C05439=1080.298,356.414,-96.423,176.101,28.139,154.837
C05440=1080.292,356.167,-96.387,176.097,28.133,154.836
C05441=1080.286,355.919,-96.351,176.094,28.128,154.835
C05442=1080.280,355.672,-96.316,176.091,28.123,154.834
C05443=1080.275,355.425,-96.280,176.087,28.117,154.833
C05444=1080.268,355.178,-96.244,176.084,28.111,154.832
C05445=1080.262,354.930,-96.209,176.081,28.106,154.831
C05446=1080.256,354.683,-96.173,176.078,28.100,154.830
C05447=1080.249,354.435,-96.137,176.074,28.095,154.829
C05448=1080.244,354.188,-96.102,176.071,28.089,154.828
C05449=1080.237,353.941,-96.067,176.068,28.083,154.827
C05450=1080.231,353.693,-96.031,176.065,28.078,154.826
C05451=1080.225,353.445,-95.995,176.061,28.073,154.825
C05452=1080.220,353.198,-95.960,176.058,28.067,154.824
C05453=1080.213,352.951,-95.925,176.055,28.062,154.823
C05454=1080.207,352.703,-95.889,176.052,28.056,154.822
C05455=1080.201,352.456,-95.853,176.048,28.051,154.821
C05456=1080.195,352.209,-95.818,176.045,28.045,154.820
C05457=1080.189,351.961,-95.783,176.041,28.040,154.820
C05458=1080.183,351.714,-95.747,176.038,28.035,154.819
C05459=1080.176,351.466,-95.712,176.034,28.029,154.818
C05460=1080.171,351.219,-95.676,176.031,28.024,154.817
C05461=1080.164,350.972,-95.641,176.028,28.019,154.816
C05462=1080.158,350.724,-95.606,176.025,28.013,154.815
C05463=1080.153,350.477,-95.571,176.022,28.008,154.814
C05464=1080.146,350.229,-95.536,176.018,28.002,154.813
C05465=1080.140,349.982,-95.500,176.015,27.997,154.812
C05466=1080.134,349.735,-95.465,176.012,27.992,154.811
C05467=1080.128,349.487,-95.430,176.009,27.987,154.810
C05468=1080.121,349.239,-95.395,176.005,27.981,154.809
C05469=1080.116,348.992,-95.360,176.002,27.976,154.808
C05470=1080.109,348.745,-95.325,175.999,27.971,154.807
C05471=1080.103,348.497,-95.290,175.995,27.965,154.807
C05472=1080.097,348.250,-95.255,175.992,27.960,154.806
C05473=1080.091,348.002,-95.219,175.989,27.955,154.805
C05474=1080.085,347.755,-95.185,175.985,27.950,154.804
C05475=1080.079,347.507,-95.149,175.982,27.944,154.803
C05476=1080.073,347.259,-95.115,175.979,27.939,154.802
C05477=1080.067,347.012,-95.080,175.976,27.934,154.801
C05478=1080.061,346.765,-95.044,175.973,27.929,154.800
C05479=1080.055,346.518,-95.010,175.970,27.924,154.799
C05480=1080.049,346.270,-94.975,175.966,27.918,154.798
C05481=1080.043,346.022,-94.940,175.963,27.913,154.797
C05482=1080.037,345.775,-94.905,175.959,27.908,154.797
C05483=1080.030,345.527,-94.870,175.956,27.903,154.796
C05484=1080.025,345.280,-94.835,175.953,27.898,154.795
C05485=1080.018,345.032,-94.801,175.950,27.893,154.794
C05486=1080.009,344.621,-94.743,175.945,27.884,154.793
C05487=1079.998,344.208,-94.686,175.939,27.876,154.791
C05488=1079.988,343.795,-94.628,175.934,27.867,154.790
C05489=1079.978,343.384,-94.570,175.928,27.858,154.788
C05490=1079.972,343.135,-94.535,175.925,27.854,154.787
C05491=1079.967,342.888,-94.501,175.922,27.848,154.786
C05492=1079.960,342.641,-94.466,175.919,27.843,154.786
C05493=1079.954,342.394,-94.432,175.916,27.839,154.785
C05494=1079.947,342.146,-94.397,175.912,27.833,154.784
C05495=1079.942,341.898,-94.363,175.909,27.828,154.783
C05496=1079.936,341.650,-94.328,175.906,27.823,154.782
C05497=1079.930,341.403,-94.294,175.903,27.818,154.781
C05498=1079.923,341.155,-94.259,175.899,27.813,154.781
C05499=1079.917,340.908,-94.225,175.896,27.808,154.780
C05500=1079.912,340.661,-94.191,175.893,27.803,154.779
C05501=1079.906,340.412,-94.156,175.890,27.798,154.778
C05502=1079.900,340.165,-94.122,175.887,27.793,154.777
C05503=1079.894,339.917,-94.087,175.884,27.788,154.776
C05504=1079.888,339.670,-94.053,175.881,27.784,154.775
C05505=1079.882,339.423,-94.019,175.877,27.778,154.775
C05506=1079.875,339.175,-93.985,175.874,27.773,154.774
C05507=1079.869,338.927,-93.951,175.871,27.768,154.773
C05508=1079.864,338.679,-93.916,175.867,27.763,154.772
C05509=1079.858,338.432,-93.882,175.864,27.758,154.771
C05510=1079.852,338.184,-93.848,175.861,27.754,154.770
C05511=1079.846,337.936,-93.813,175.858,27.748,154.770
C05512=1079.840,337.689,-93.779,175.855,27.744,154.769
C05513=1079.834,337.441,-93.746,175.852,27.739,154.768
C05514=1079.828,337.193,-93.712,175.849,27.734,154.767
C05515=1079.822,336.946,-93.678,175.846,27.729,154.766
C05516=1079.816,336.699,-93.643,175.843,27.724,154.766
C05517=1079.809,336.451,-93.609,175.839,27.720,154.765
C05518=1079.804,336.203,-93.575,175.836,27.715,154.764
C05519=1079.797,335.956,-93.542,175.833,27.710,154.763
C05520=1079.791,335.708,-93.508,175.830,27.705,154.762
C05521=1079.785,335.461,-93.474,175.827,27.700,154.762
C05522=1079.779,335.213,-93.440,175.824,27.695,154.761
C05523=1079.773,334.965,-93.406,175.821,27.691,154.760
C05524=1079.767,334.717,-93.372,175.818,27.685,154.759
C05525=1079.761,334.470,-93.338,175.815,27.681,154.758
C05526=1079.756,334.222,-93.305,175.811,27.676,154.758
C05527=1079.749,333.974,-93.270,175.807,27.671,154.757
C05528=1079.744,333.726,-93.237,175.804,27.666,154.756
C05529=1079.737,333.479,-93.203,175.801,27.662,154.755
C05530=1079.731,333.232,-93.169,175.798,27.656,154.754
C05531=1079.726,332.984,-93.136,175.795,27.652,154.754
C05532=1079.719,332.736,-93.102,175.792,27.647,154.753
C05533=1079.714,332.488,-93.068,175.789,27.642,154.752
C05534=1079.708,332.241,-93.034,175.786,27.638,154.751
C05535=1079.702,331.993,-93.001,175.783,27.633,154.750
C05536=1079.696,331.746,-92.967,175.780,27.628,154.750
C05537=1079.690,331.498,-92.934,175.777,27.624,154.749
C05538=1079.679,331.080,-92.877,175.772,27.615,154.748
C05539=1079.669,330.662,-92.821,175.766,27.608,154.746
C05540=1079.659,330.245,-92.765,175.760,27.600,154.745
C05541=1079.648,329.827,-92.708,175.756,27.592,154.744
C05542=1079.642,329.579,-92.674,175.753,27.588,154.743
C05543=1079.636,329.331,-92.642,175.750,27.583,154.742
C05544=1079.630,329.084,-92.608,175.746,27.579,154.742
C05545=1079.624,328.836,-92.575,175.743,27.574,154.741
C05546=1079.618,328.588,-92.542,175.740,27.569,154.740
C05547=1079.612,328.341,-92.509,175.737,27.565,154.739
C05548=1079.606,328.092,-92.475,175.734,27.560,154.739
C05549=1079.599,327.845,-92.442,175.731,27.555,154.738
C05550=1079.594,327.597,-92.408,175.728,27.551,154.737
C05551=1079.587,327.350,-92.376,175.725,27.546,154.736
C05552=1079.582,327.102,-92.342,175.721,27.542,154.736
C05553=1079.575,326.854,-92.310,175.718,27.537,154.735
C05554=1079.570,326.606,-92.276,175.715,27.533,154.734
C05555=1079.564,326.359,-92.243,175.712,27.528,154.733
C05556=1079.558,326.112,-92.209,175.709,27.523,154.733
C05557=1079.551,325.863,-92.176,175.707,27.519,154.732
C05558=1079.545,325.615,-92.143,175.704,27.515,154.731
C05559=1079.539,325.368,-92.110,175.700,27.510,154.730
C05560=1079.533,325.120,-92.077,175.697,27.506,154.730
C05561=1079.527,324.872,-92.044,175.694,27.501,154.729
C05562=1079.521,324.625,-92.011,175.691,27.497,154.728
C05563=1079.515,324.377,-91.978,175.688,27.492,154.728
C05564=1079.509,324.129,-91.945,175.685,27.487,154.727
C05565=1079.503,323.881,-91.912,175.682,27.483,154.726
C05566=1079.497,323.633,-91.880,175.678,27.478,154.725
C05567=1079.491,323.385,-91.847,175.676,27.474,154.725
C05568=1079.486,323.138,-91.814,175.673,27.469,154.724
C05569=1079.479,322.890,-91.781,175.670,27.465,154.723
C05570=1079.474,322.642,-91.748,175.667,27.460,154.723
C05571=1079.467,322.394,-91.715,175.664,27.456,154.722
C05572=1079.461,322.147,-91.682,175.660,27.451,154.721
C05573=1079.457,321.899,-91.650,175.657,27.447,154.720
C05574=1079.450,321.651,-91.617,175.654,27.442,154.720
C05575=1079.445,321.404,-91.584,175.651,27.438,154.719
C05576=1079.438,321.156,-91.551,175.649,27.434,154.718
C05577=1079.432,320.908,-91.518,175.646,27.429,154.717
C05578=1079.427,320.660,-91.486,175.643,27.425,154.717
C05579=1079.421,320.412,-91.453,175.639,27.420,154.716
C05580=1079.414,320.165,-91.420,175.636,27.416,154.715
C05581=1079.409,319.916,-91.388,175.633,27.411,154.715
C05582=1079.403,319.669,-91.355,175.630,27.407,154.714
C05583=1079.397,319.422,-91.323,175.628,27.402,154.713
C05584=1079.392,319.173,-91.290,175.625,27.398,154.713
C05585=1079.386,318.925,-91.257,175.622,27.393,154.712
C05586=1079.379,318.678,-91.225,175.618,27.389,154.711
C05587=1079.374,318.430,-91.193,175.615,27.384,154.710
C05588=1079.368,318.182,-91.160,175.612,27.380,154.710
C05589=1079.362,317.934,-91.128,175.610,27.376,154.709
C05590=1079.357,317.723,-91.099,175.607,27.372,154.708
C05591=1079.353,317.510,-91.072,175.605,27.368,154.708
C05592=1079.347,317.297,-91.044,175.602,27.364,154.707
C05593=1079.342,317.086,-91.015,175.599,27.360,154.707
C05594=1079.337,316.874,-90.988,175.597,27.356,154.706
C05595=1079.332,316.662,-90.961,175.594,27.353,154.705
C05596=1079.328,316.449,-90.933,175.592,27.349,154.705
C05597=1079.323,316.238,-90.905,175.589,27.345,154.704
C05598=1079.317,315.989,-90.873,175.587,27.341,154.703
C05599=1079.311,315.741,-90.841,175.584,27.337,154.703
C05600=1079.306,315.494,-90.808,175.580,27.332,154.702
C05601=1079.300,315.246,-90.776,175.577,27.327,154.701
C05602=1079.294,314.998,-90.743,175.574,27.323,154.701
C05603=1079.288,314.751,-90.711,175.572,27.319,154.700
C05604=1079.282,314.502,-90.679,175.569,27.314,154.699
C05605=1079.276,314.255,-90.646,175.566,27.310,154.699
C05606=1079.270,314.007,-90.614,175.562,27.306,154.698
C05607=1079.264,313.758,-90.582,175.559,27.302,154.697
C05608=1079.258,313.511,-90.551,175.556,27.297,154.697
C05609=1079.251,313.264,-90.519,175.554,27.293,154.696
C05610=1079.245,313.015,-90.487,175.551,27.289,154.695
C05611=1079.239,312.767,-90.455,175.548,27.285,154.695
C05612=1079.233,312.519,-90.422,175.544,27.281,154.694
C05613=1079.228,312.272,-90.391,175.541,27.276,154.694
C05614=1079.221,312.024,-90.359,175.539,27.272,154.693
C05615=1079.215,311.776,-90.327,175.536,27.268,154.692
C05616=1079.210,311.529,-90.295,175.533,27.264,154.692
C05617=1079.204,311.280,-90.263,175.530,27.260,154.691
C05618=1079.198,311.032,-90.231,175.527,27.256,154.690
C05619=1079.191,310.784,-90.200,175.524,27.251,154.690
C05620=1079.186,310.537,-90.168,175.521,27.247,154.689
C05621=1079.180,310.288,-90.136,175.518,27.243,154.688
C05622=1079.174,310.040,-90.104,175.515,27.238,154.688
C05623=1079.168,309.793,-90.073,175.512,27.234,154.687
C05624=1079.162,309.545,-90.041,175.509,27.230,154.686
C05625=1079.156,309.297,-90.009,175.506,27.226,154.686
C05626=1079.150,309.049,-89.977,175.503,27.222,154.685
C05627=1079.143,308.801,-89.946,175.501,27.218,154.684
C05628=1079.138,308.554,-89.914,175.498,27.213,154.684
C05629=1079.132,308.305,-89.882,175.494,27.209,154.683
C05630=1079.127,308.058,-89.850,175.491,27.205,154.682
C05631=1079.120,307.810,-89.819,175.488,27.201,154.682
C05632=1079.114,307.562,-89.787,175.486,27.197,154.681
C05633=1079.109,307.314,-89.755,175.483,27.193,154.681
C05634=1079.102,307.066,-89.724,175.480,27.188,154.680
C05635=1079.096,306.819,-89.692,175.476,27.184,154.679
C05636=1079.091,306.570,-89.661,175.474,27.180,154.679
C05637=1079.085,306.323,-89.630,175.471,27.176,154.678
C05638=1079.079,306.075,-89.598,175.468,27.172,154.677
C05639=1079.073,305.827,-89.566,175.465,27.167,154.677
C05640=1079.067,305.579,-89.535,175.463,27.163,154.676
C05641=1079.061,305.331,-89.504,175.459,27.159,154.675
C05642=1079.056,305.083,-89.472,175.456,27.155,154.675
C05643=1079.049,304.836,-89.440,175.454,27.151,154.674
C05644=1079.043,304.587,-89.408,175.451,27.147,154.674
C05645=1079.038,304.339,-89.378,175.448,27.143,154.673
C05646=1079.032,304.129,-89.351,175.445,27.139,154.672
C05647=1079.028,303.919,-89.324,175.443,27.136,154.672
C05648=1079.023,303.708,-89.297,175.441,27.132,154.671
C05649=1079.018,303.497,-89.271,175.437,27.128,154.671
C05650=1079.013,303.287,-89.244,175.435,27.125,154.670
C05651=1079.008,303.076,-89.217,175.433,27.121,154.670
C05652=1079.003,302.866,-89.192,175.431,27.118,154.669
C05653=1078.998,302.655,-89.164,175.428,27.115,154.669
C05654=1078.993,302.407,-89.133,175.425,27.110,154.668
C05655=1078.986,302.159,-89.102,175.422,27.106,154.667
C05656=1078.981,301.911,-89.071,175.420,27.102,154.667
C05657=1078.975,301.663,-89.040,175.417,27.098,154.666
C05658=1078.970,301.415,-89.009,175.413,27.094,154.666
C05659=1078.964,301.167,-88.977,175.411,27.090,154.665
C05660=1078.958,300.919,-88.946,175.408,27.086,154.664
C05661=1078.952,300.671,-88.915,175.405,27.081,154.664
C05662=1078.947,300.423,-88.884,175.403,27.077,154.663
C05663=1078.941,300.175,-88.852,175.400,27.073,154.662
C05664=1078.935,299.927,-88.822,175.396,27.069,154.662
C05665=1078.929,299.680,-88.790,175.394,27.065,154.661
C05666=1078.923,299.431,-88.759,175.391,27.061,154.661
C05667=1078.918,299.184,-88.728,175.388,27.057,154.660
C05668=1078.912,298.936,-88.697,175.385,27.052,154.659
C05669=1078.907,298.688,-88.666,175.383,27.048,154.659
C05670=1078.901,298.440,-88.634,175.379,27.044,154.658
C05671=1078.895,298.192,-88.604,175.377,27.040,154.657
C05672=1078.890,297.944,-88.573,175.374,27.036,154.657
C05673=1078.884,297.697,-88.542,175.371,27.032,154.656
C05674=1078.877,297.448,-88.511,175.369,27.028,154.656
C05675=1078.872,297.200,-88.480,175.365,27.024,154.655
C05676=1078.866,296.952,-88.450,175.362,27.020,154.654
C05677=1078.860,296.704,-88.419,175.360,27.016,154.654
C05678=1078.855,296.456,-88.388,175.357,27.012,154.653
C05679=1078.849,296.208,-88.357,175.354,27.008,154.652
C05680=1078.842,295.960,-88.327,175.351,27.004,154.652
C05681=1078.836,295.712,-88.296,175.348,27.000,154.651
C05682=1078.831,295.464,-88.265,175.345,26.996,154.651
C05683=1078.825,295.215,-88.235,175.343,26.992,154.650
C05684=1078.819,294.968,-88.204,175.340,26.988,154.649
C05685=1078.813,294.720,-88.173,175.337,26.984,154.649
C05686=1078.807,294.472,-88.143,175.334,26.980,154.648
C05687=1078.802,294.224,-88.112,175.331,26.976,154.648
C05688=1078.796,293.976,-88.081,175.328,26.972,154.647
C05689=1078.790,293.728,-88.051,175.326,26.968,154.647
C05690=1078.784,293.480,-88.020,175.323,26.964,154.646
C05691=1078.778,293.232,-87.990,175.320,26.960,154.645
C05692=1078.772,292.984,-87.959,175.317,26.956,154.645
C05693=1078.766,292.736,-87.929,175.314,26.952,154.644
C05694=1078.761,292.488,-87.898,175.312,26.948,154.644
C05695=1078.755,292.240,-87.868,175.309,26.944,154.643
C05696=1078.749,291.991,-87.837,175.306,26.940,154.642
C05697=1078.743,291.744,-87.807,175.303,26.936,154.642
C05698=1078.737,291.496,-87.776,175.300,26.932,154.641
C05699=1078.732,291.247,-87.747,175.298,26.928,154.641
C05700=1078.726,291.000,-87.716,175.295,26.924,154.640
C05701=1078.719,290.751,-87.686,175.292,26.920,154.639
C05702=1078.710,290.344,-87.636,175.288,26.914,154.639
C05703=1078.700,289.938,-87.586,175.283,26.907,154.638
C05704=1078.691,289.531,-87.536,175.279,26.901,154.637
C05705=1078.682,289.124,-87.487,175.274,26.894,154.636
C05706=1078.675,288.876,-87.456,175.271,26.891,154.635
C05707=1078.670,288.628,-87.427,175.268,26.887,154.635
C05708=1078.664,288.380,-87.396,175.265,26.883,154.634
C05709=1078.658,288.132,-87.366,175.262,26.879,154.633
C05710=1078.652,287.884,-87.337,175.260,26.875,154.633
C05711=1078.646,287.636,-87.307,175.257,26.871,154.632
C05712=1078.640,287.388,-87.276,175.254,26.868,154.632
C05713=1078.634,287.139,-87.246,175.251,26.863,154.631
C05714=1078.628,286.891,-87.216,175.249,26.860,154.631
C05715=1078.623,286.643,-87.186,175.246,26.856,154.630
C05716=1078.617,286.395,-87.156,175.243,26.852,154.629
C05717=1078.611,286.147,-87.126,175.240,26.848,154.629
C05718=1078.605,285.899,-87.097,175.237,26.844,154.628
C05719=1078.599,285.651,-87.066,175.235,26.840,154.628
C05720=1078.594,285.403,-87.037,175.232,26.836,154.627
C05721=1078.588,285.155,-87.006,175.230,26.832,154.627
C05722=1078.582,284.906,-86.977,175.226,26.828,154.626
C05723=1078.577,284.659,-86.946,175.224,26.825,154.625
C05724=1078.570,284.410,-86.917,175.221,26.821,154.625
C05725=1078.564,284.163,-86.887,175.218,26.817,154.624
C05726=1078.559,283.914,-86.857,175.216,26.813,154.624
C05727=1078.553,283.666,-86.827,175.213,26.809,154.623
C05728=1078.548,283.418,-86.797,175.210,26.805,154.623
C05729=1078.541,283.170,-86.767,175.207,26.801,154.622
C05730=1078.536,282.922,-86.738,175.205,26.798,154.621
C05731=1078.530,282.674,-86.708,175.202,26.794,154.621
C05732=1078.524,282.426,-86.678,175.200,26.790,154.620
C05733=1078.519,282.177,-86.648,175.196,26.786,154.620
C05734=1078.513,281.929,-86.619,175.194,26.782,154.619
C05735=1078.507,281.681,-86.589,175.191,26.778,154.619
C05736=1078.501,281.433,-86.559,175.189,26.774,154.618
C05737=1078.496,281.184,-86.529,175.186,26.770,154.617
C05738=1078.489,280.937,-86.500,175.182,26.766,154.617
C05739=1078.484,280.688,-86.470,175.180,26.763,154.616
C05740=1078.478,280.440,-86.440,175.177,26.758,154.616
C05741=1078.472,280.192,-86.411,175.175,26.755,154.615
C05742=1078.466,279.943,-86.382,175.172,26.751,154.615
C05743=1078.460,279.696,-86.352,175.169,26.747,154.614
C05744=1078.454,279.447,-86.322,175.166,26.743,154.614
C05745=1078.449,279.199,-86.293,175.164,26.740,154.613
C05746=1078.442,278.951,-86.264,175.161,26.736,154.613
C05747=1078.437,278.702,-86.234,175.159,26.732,154.612
C05748=1078.431,278.454,-86.205,175.155,26.728,154.611
C05749=1078.425,278.206,-86.175,175.153,26.724,154.611
C05750=1078.420,277.959,-86.145,175.150,26.720,154.610
C05751=1078.414,277.711,-86.116,175.148,26.717,154.610
C05752=1078.408,277.462,-86.087,175.145,26.713,154.609
C05753=1078.402,277.214,-86.058,175.142,26.709,154.609
C05754=1078.393,276.817,-86.011,175.138,26.703,154.608
C05755=1078.384,276.419,-85.964,175.134,26.697,154.607
C05756=1078.374,276.023,-85.917,175.129,26.691,154.606
C05757=1078.365,275.626,-85.870,175.125,26.685,154.605
C05758=1078.359,275.378,-85.841,175.122,26.681,154.605
C05759=1078.353,275.130,-85.812,175.120,26.677,154.604
C05760=1078.347,274.881,-85.782,175.117,26.673,154.603
C05761=1078.341,274.633,-85.753,175.115,26.670,154.603
C05762=1078.337,274.385,-85.725,175.112,26.666,154.602
C05763=1078.330,274.137,-85.696,175.109,26.662,154.602
C05764=1078.325,273.888,-85.666,175.106,26.658,154.601
C05765=1078.319,273.640,-85.637,175.104,26.654,154.601
C05766=1078.312,273.392,-85.608,175.101,26.651,154.600
C05767=1078.307,273.144,-85.579,175.099,26.647,154.600
C05768=1078.301,272.896,-85.550,175.095,26.643,154.599
C05769=1078.296,272.647,-85.521,175.093,26.639,154.599
C05770=1078.290,272.399,-85.492,175.090,26.635,154.598
C05771=1078.283,272.151,-85.463,175.088,26.632,154.597
C05772=1078.278,271.903,-85.435,175.085,26.628,154.597
C05773=1078.273,271.654,-85.405,175.082,26.624,154.596
C05774=1078.266,271.406,-85.376,175.080,26.621,154.596
C05775=1078.260,271.157,-85.348,175.077,26.617,154.595
C05776=1078.255,270.909,-85.318,175.075,26.613,154.595
C05777=1078.249,270.662,-85.289,175.072,26.609,154.594
C05778=1078.243,270.413,-85.261,175.069,26.605,154.594
C05779=1078.238,270.164,-85.231,175.066,26.602,154.593
C05780=1078.232,269.916,-85.202,175.064,26.598,154.593
C05781=1078.226,269.668,-85.174,175.061,26.594,154.592
C05782=1078.220,269.420,-85.145,175.059,26.591,154.592
C05783=1078.214,269.172,-85.116,175.056,26.587,154.591
C05784=1078.209,268.924,-85.088,175.053,26.583,154.590
C05785=1078.203,268.675,-85.059,175.051,26.579,154.590
C05786=1078.197,268.427,-85.030,175.048,26.575,154.589
C05787=1078.191,268.179,-85.001,175.046,26.572,154.589
C05788=1078.185,267.930,-84.973,175.042,26.568,154.588
C05789=1078.179,267.682,-84.944,175.040,26.564,154.588
C05790=1078.174,267.433,-84.916,175.037,26.561,154.587
C05791=1078.168,267.186,-84.887,175.035,26.557,154.587
C05792=1078.162,266.937,-84.859,175.033,26.553,154.586
C05793=1078.156,266.689,-84.829,175.029,26.550,154.586
C05794=1078.151,266.441,-84.802,175.027,26.545,154.585
C05795=1078.145,266.192,-84.773,175.024,26.542,154.585
C05796=1078.138,265.944,-84.744,175.022,26.538,154.584
C05797=1078.133,265.696,-84.716,175.020,26.535,154.584
C05798=1078.128,265.447,-84.687,175.016,26.531,154.583
C05799=1078.122,265.199,-84.658,175.014,26.527,154.583
C05800=1078.116,264.951,-84.630,175.011,26.523,154.582
C05801=1078.110,264.703,-84.601,175.009,26.520,154.581
C05802=1078.104,264.454,-84.573,175.007,26.516,154.581
C05803=1078.099,264.206,-84.545,175.004,26.512,154.580
C05804=1078.093,263.957,-84.517,175.001,26.508,154.580
C05805=1078.087,263.710,-84.488,174.998,26.504,154.579
C05806=1078.077,263.315,-84.443,174.994,26.499,154.579
C05807=1078.068,262.921,-84.399,174.991,26.493,154.578
C05808=1078.059,262.527,-84.354,174.986,26.487,154.577
C05809=1078.049,262.134,-84.309,174.982,26.481,154.576
C05810=1078.043,261.885,-84.281,174.979,26.478,154.576
C05811=1078.038,261.637,-84.253,174.977,26.474,154.575
C05812=1078.031,261.389,-84.225,174.974,26.470,154.575
C05813=1078.025,261.140,-84.197,174.971,26.467,154.574
C05814=1078.020,260.892,-84.168,174.969,26.463,154.573
C05815=1078.014,260.644,-84.140,174.966,26.459,154.573
C05816=1078.008,260.396,-84.112,174.964,26.456,154.573
C05817=1078.002,260.147,-84.084,174.961,26.453,154.572
C05818=1077.996,259.898,-84.056,174.958,26.449,154.572
C05819=1077.990,259.650,-84.028,174.956,26.445,154.571
C05820=1077.984,259.402,-83.999,174.954,26.442,154.570
C05821=1077.978,259.154,-83.972,174.951,26.438,154.570
C05822=1077.972,258.905,-83.944,174.948,26.434,154.569
C05823=1077.967,258.657,-83.916,174.945,26.430,154.569
C05824=1077.961,258.408,-83.887,174.943,26.427,154.568
C05825=1077.955,258.161,-83.860,174.941,26.423,154.568
C05826=1077.949,257.912,-83.832,174.938,26.419,154.567
C05827=1077.944,257.664,-83.804,174.935,26.416,154.567
C05828=1077.938,257.415,-83.775,174.933,26.412,154.566
C05829=1077.932,257.167,-83.749,174.930,26.408,154.566
C05830=1077.926,256.918,-83.720,174.928,26.405,154.565
C05831=1077.921,256.670,-83.692,174.926,26.401,154.565
C05832=1077.915,256.421,-83.664,174.922,26.397,154.564
C05833=1077.909,256.173,-83.637,174.920,26.394,154.564
C05834=1077.903,255.925,-83.608,174.918,26.390,154.563
C05835=1077.898,255.677,-83.580,174.915,26.386,154.563
C05836=1077.891,255.428,-83.553,174.913,26.383,154.562
C05837=1077.886,255.179,-83.525,174.910,26.379,154.562
C05838=1077.880,254.931,-83.497,174.907,26.375,154.561
C05839=1077.874,254.683,-83.470,174.905,26.372,154.561
C05840=1077.868,254.434,-83.442,174.903,26.368,154.560
C05841=1077.863,254.186,-83.414,174.900,26.364,154.560
C05842=1077.857,253.938,-83.387,174.897,26.360,154.559
C05843=1077.851,253.689,-83.358,174.895,26.357,154.559
C05844=1077.846,253.440,-83.331,174.892,26.353,154.558
C05845=1077.839,253.192,-83.304,174.890,26.349,154.557
C05846=1077.834,252.944,-83.276,174.888,26.346,154.557
C05847=1077.829,252.695,-83.248,174.885,26.342,154.556
C05848=1077.822,252.447,-83.221,174.882,26.338,154.556
C05849=1077.817,252.199,-83.193,174.880,26.335,154.555
C05850=1077.812,251.950,-83.165,174.877,26.331,154.555
C05851=1077.805,251.702,-83.138,174.875,26.327,154.554
C05852=1077.800,251.453,-83.110,174.873,26.324,154.554
C05853=1077.795,251.205,-83.082,174.869,26.320,154.553
C05854=1077.788,250.956,-83.055,174.867,26.316,154.553
C05855=1077.783,250.708,-83.027,174.865,26.313,154.552
C05856=1077.777,250.460,-83.000,174.862,26.309,154.552
C05857=1077.771,250.211,-82.973,174.860,26.305,154.551
C05858=1077.763,249.815,-82.928,174.856,26.299,154.550
C05859=1077.753,249.418,-82.885,174.852,26.293,154.549
C05860=1077.744,249.021,-82.841,174.848,26.287,154.549
C05861=1077.735,248.625,-82.798,174.844,26.281,154.548
C05862=1077.729,248.376,-82.770,174.842,26.278,154.547
C05863=1077.724,248.128,-82.743,174.840,26.274,154.547
C05864=1077.718,247.880,-82.715,174.836,26.270,154.546
C05865=1077.713,247.631,-82.688,174.834,26.267,154.546
C05866=1077.707,247.382,-82.661,174.832,26.263,154.545
C05867=1077.701,247.134,-82.633,174.829,26.259,154.545
C05868=1077.696,246.886,-82.606,174.827,26.255,154.544
C05869=1077.690,246.637,-82.579,174.825,26.252,154.544
C05870=1077.684,246.389,-82.551,174.822,26.248,154.543
C05871=1077.678,246.140,-82.525,174.819,26.244,154.543
C05872=1077.673,245.892,-82.497,174.817,26.241,154.542
C05873=1077.667,245.644,-82.470,174.815,26.237,154.542
C05874=1077.661,245.395,-82.443,174.813,26.234,154.541
C05875=1077.656,245.146,-82.416,174.809,26.230,154.541
C05876=1077.650,244.898,-82.389,174.807,26.226,154.540
C05877=1077.644,244.650,-82.362,174.805,26.223,154.539
C05878=1077.639,244.401,-82.334,174.802,26.219,154.539
C05879=1077.632,244.152,-82.307,174.800,26.215,154.538
C05880=1077.627,243.904,-82.281,174.798,26.211,154.538
C05881=1077.622,243.655,-82.253,174.795,26.208,154.537
C05882=1077.616,243.407,-82.227,174.792,26.204,154.537
C05883=1077.610,243.159,-82.199,174.790,26.200,154.536
C05884=1077.604,242.910,-82.172,174.788,26.197,154.536
C05885=1077.598,242.661,-82.145,174.786,26.193,154.535
C05886=1077.593,242.413,-82.119,174.783,26.189,154.535
C05887=1077.587,242.165,-82.092,174.780,26.186,154.534
C05888=1077.581,241.916,-82.065,174.778,26.183,154.534
C05889=1077.575,241.667,-82.038,174.776,26.179,154.533
C05890=1077.570,241.419,-82.011,174.773,26.175,154.533
C05891=1077.564,241.170,-81.984,174.771,26.171,154.532
C05892=1077.558,240.922,-81.958,174.768,26.168,154.532
C05893=1077.552,240.674,-81.931,174.766,26.164,154.531
C05894=1077.547,240.425,-81.904,174.763,26.160,154.531
C05895=1077.540,240.176,-81.877,174.761,26.157,154.530
C05896=1077.534,239.928,-81.851,174.759,26.153,154.530
C05897=1077.529,239.679,-81.824,174.756,26.150,154.529
C05898=1077.524,239.431,-81.797,174.754,26.146,154.529
C05899=1077.518,239.182,-81.770,174.751,26.142,154.528
C05900=1077.512,238.934,-81.744,174.749,26.139,154.528
C05901=1077.506,238.685,-81.717,174.747,26.135,154.527
C05902=1077.500,238.437,-81.690,174.744,26.132,154.527
C05903=1077.494,238.188,-81.663,174.741,26.128,154.526
C05904=1077.489,237.939,-81.637,174.739,26.124,154.526
C05905=1077.483,237.691,-81.611,174.737,26.121,154.525
C05906=1077.477,237.443,-81.584,174.735,26.117,154.525
C05907=1077.471,237.194,-81.557,174.733,26.113,154.524
C05908=1077.466,236.946,-81.531,174.729,26.110,154.524
C05909=1077.460,236.698,-81.504,174.727,26.106,154.523
C05910=1077.450,236.293,-81.461,174.724,26.100,154.522
C05911=1077.441,235.891,-81.418,174.720,26.094,154.521
C05912=1077.432,235.487,-81.376,174.715,26.088,154.521
C05913=1077.423,235.085,-81.333,174.712,26.082,154.520
C05914=1077.417,234.836,-81.306,174.709,26.079,154.519
C05915=1077.412,234.587,-81.280,174.707,26.075,154.519
C05916=1077.406,234.339,-81.253,174.705,26.071,154.518
C05917=1077.400,234.091,-81.227,174.703,26.068,154.518
C05918=1077.395,233.842,-81.201,174.700,26.064,154.517
C05919=1077.389,233.593,-81.174,174.698,26.060,154.517
C05920=1077.383,233.345,-81.147,174.695,26.057,154.516
C05921=1077.377,233.095,-81.121,174.693,26.053,154.516
C05922=1077.371,232.847,-81.094,174.691,26.050,154.515
C05923=1077.366,232.598,-81.069,174.688,26.046,154.515
C05924=1077.360,232.350,-81.043,174.686,26.042,154.514
C05925=1077.354,232.102,-81.016,174.684,26.039,154.514
C05926=1077.349,231.853,-80.990,174.681,26.035,154.513
C05927=1077.343,231.605,-80.964,174.679,26.032,154.513
C05928=1077.337,231.356,-80.938,174.676,26.028,154.512
C05929=1077.332,231.107,-80.911,174.674,26.024,154.512
C05930=1077.326,230.858,-80.885,174.672,26.020,154.511
C05931=1077.320,230.610,-80.859,174.670,26.017,154.511
C05932=1077.314,230.361,-80.833,174.667,26.013,154.510
C05933=1077.308,230.113,-80.807,174.665,26.010,154.510
C05934=1077.303,229.864,-80.781,174.662,26.006,154.509
C05935=1077.296,229.616,-80.755,174.660,26.002,154.509
C05936=1077.291,229.367,-80.729,174.658,25.998,154.508
C05937=1077.285,229.118,-80.703,174.656,25.995,154.508
C05938=1077.279,228.870,-80.677,174.653,25.992,154.507
C05939=1077.273,228.621,-80.651,174.651,25.988,154.507
C05940=1077.268,228.372,-80.625,174.648,25.984,154.506
C05941=1077.261,228.124,-80.599,174.646,25.981,154.506
C05942=1077.256,227.875,-80.573,174.644,25.977,154.505
C05943=1077.251,227.626,-80.547,174.642,25.973,154.504
C05944=1077.245,227.379,-80.521,174.639,25.970,154.504
C05945=1077.239,227.130,-80.495,174.637,25.966,154.503
C05946=1077.234,226.881,-80.469,174.635,25.963,154.503
C05947=1077.227,226.633,-80.443,174.632,25.959,154.503
C05948=1077.222,226.384,-80.417,174.630,25.955,154.502
C05949=1077.215,226.135,-80.392,174.628,25.952,154.502
C05950=1077.210,225.886,-80.366,174.625,25.948,154.501
C05951=1077.204,225.638,-80.339,174.623,25.945,154.500
C05952=1077.199,225.390,-80.314,174.621,25.941,154.500
C05953=1077.193,225.141,-80.288,174.619,25.937,154.499
C05954=1077.187,224.892,-80.263,174.616,25.933,154.499
C05955=1077.182,224.643,-80.237,174.614,25.930,154.498
C05956=1077.176,224.395,-80.211,174.611,25.926,154.498
C05957=1077.170,224.146,-80.185,174.609,25.922,154.497
C05958=1077.165,223.898,-80.160,174.607,25.919,154.497
C05959=1077.158,223.649,-80.134,174.605,25.915,154.496
C05960=1077.153,223.400,-80.108,174.603,25.912,154.496
C05961=1077.148,223.151,-80.082,174.601,25.908,154.495
C05962=1077.138,222.740,-80.040,174.596,25.902,154.494
C05963=1077.129,222.328,-79.998,174.592,25.896,154.494
C05964=1077.119,221.917,-79.956,174.589,25.890,154.493
C05965=1077.110,221.506,-79.913,174.585,25.884,154.492
C05966=1077.104,221.257,-79.888,174.583,25.881,154.491
C05967=1077.098,221.008,-79.862,174.581,25.877,154.491
C05968=1077.092,220.759,-79.836,174.579,25.873,154.490
C05969=1077.086,220.510,-79.811,174.577,25.870,154.490
C05970=1077.081,220.262,-79.786,174.573,25.866,154.489
C05971=1077.075,220.013,-79.760,174.571,25.862,154.489
C05972=1077.069,219.765,-79.735,174.569,25.858,154.488
C05973=1077.063,219.516,-79.709,174.567,25.855,154.488
C05974=1077.058,219.268,-79.684,174.565,25.851,154.487
C05975=1077.052,219.019,-79.658,174.563,25.848,154.487
C05976=1077.045,218.770,-79.633,174.560,25.844,154.486
C05977=1077.040,218.521,-79.608,174.558,25.841,154.486
C05978=1077.035,218.273,-79.583,174.556,25.837,154.485
C05979=1077.028,218.024,-79.558,174.554,25.833,154.485
C05980=1077.023,217.775,-79.532,174.551,25.830,154.484
C05981=1077.017,217.527,-79.507,174.549,25.826,154.484
C05982=1077.011,217.279,-79.481,174.547,25.822,154.483
C05983=1077.006,217.029,-79.456,174.544,25.819,154.483
C05984=1077.000,216.780,-79.431,174.542,25.815,154.482
C05985=1076.994,216.532,-79.406,174.540,25.811,154.482
C05986=1076.988,216.284,-79.380,174.538,25.808,154.481
C05987=1076.983,216.034,-79.355,174.536,25.804,154.481
C05988=1076.977,215.786,-79.330,174.534,25.800,154.480
C05989=1076.971,215.537,-79.305,174.532,25.797,154.480
C05990=1076.966,215.289,-79.279,174.529,25.793,154.479
C05991=1076.960,215.040,-79.255,174.527,25.790,154.479
C05992=1076.954,214.791,-79.229,174.525,25.786,154.478
C05993=1076.948,214.543,-79.204,174.522,25.782,154.478
C05994=1076.943,214.294,-79.179,174.520,25.778,154.477
C05995=1076.937,214.045,-79.154,174.518,25.775,154.477
C05996=1076.931,213.797,-79.129,174.516,25.771,154.476
C05997=1076.926,213.548,-79.104,174.513,25.767,154.475
C05998=1076.921,213.299,-79.079,174.511,25.764,154.475
C05999=1076.914,213.051,-79.053,174.509,25.760,154.474
C06000=1076.909,212.801,-79.029,174.507,25.757,154.474
C06001=1076.903,212.553,-79.004,174.505,25.753,154.474
C06002=1076.897,212.304,-78.979,174.503,25.750,154.473
C06003=1076.891,212.056,-78.954,174.501,25.746,154.472
C06004=1076.886,211.807,-78.930,174.498,25.742,154.472
C06005=1076.879,211.558,-78.904,174.496,25.739,154.471
C06006=1076.875,211.309,-78.879,174.494,25.735,154.471
C06007=1076.869,211.061,-78.854,174.492,25.731,154.470
C06008=1076.863,210.812,-78.830,174.490,25.728,154.470
C06009=1076.857,210.563,-78.804,174.488,25.724,154.469
C06010=1076.852,210.315,-78.780,174.486,25.720,154.469
C06011=1076.846,210.066,-78.755,174.483,25.717,154.468
C06012=1076.840,209.817,-78.730,174.480,25.713,154.468
C06013=1076.834,209.569,-78.705,174.478,25.709,154.467
C06014=1076.825,209.161,-78.665,174.475,25.703,154.466
C06015=1076.816,208.754,-78.624,174.472,25.698,154.466
C06016=1076.806,208.347,-78.584,174.468,25.692,154.465
C06017=1076.796,207.939,-78.543,174.465,25.686,154.464
C06018=1076.773,206.902,-78.443,174.351,25.626,154.464
C06019=1076.768,206.653,-78.419,174.349,25.623,154.464
C06020=1076.761,206.404,-78.395,174.347,25.620,154.464
C06021=1076.756,206.156,-78.370,174.344,25.618,154.464
C06022=1076.750,205.907,-78.346,174.343,25.615,154.463
C06023=1076.745,205.658,-78.323,174.341,25.613,154.463
C06024=1076.739,205.409,-78.299,174.338,25.610,154.463
C06025=1076.734,205.160,-78.274,174.336,25.607,154.462
C06026=1076.728,204.912,-78.250,174.334,25.604,154.462
C06027=1076.722,204.664,-78.226,174.331,25.602,154.462
C06028=1076.717,204.414,-78.202,174.329,25.599,154.462
C06029=1076.711,204.165,-78.178,174.326,25.596,154.461
C06030=1076.705,203.917,-78.155,174.324,25.594,154.461
C06031=1076.700,203.668,-78.130,174.322,25.591,154.461
C06032=1076.695,203.419,-78.107,174.319,25.588,154.460
C06033=1076.688,203.170,-78.083,174.317,25.586,154.460
C06034=1076.683,202.921,-78.058,174.315,25.583,154.460
C06035=1076.678,202.673,-78.034,174.312,25.580,154.459
C06036=1076.672,202.424,-78.011,174.310,25.577,154.459
C06037=1076.667,202.175,-77.987,174.308,25.575,154.459
C06038=1076.660,201.926,-77.963,174.306,25.572,154.459
C06039=1076.654,201.677,-77.940,174.304,25.570,154.458
C06040=1076.649,201.429,-77.916,174.301,25.567,154.458
C06041=1076.643,201.180,-77.893,174.299,25.565,154.458
C06042=1076.637,200.931,-77.868,174.297,25.562,154.457
C06043=1076.631,200.682,-77.845,174.294,25.559,154.457
C06044=1076.626,200.433,-77.821,174.292,25.556,154.457
C06045=1076.620,200.185,-77.797,174.290,25.554,154.457
C06046=1076.615,199.936,-77.774,174.287,25.551,154.456
C06047=1076.609,199.687,-77.750,174.285,25.549,154.456
C06048=1076.603,199.438,-77.727,174.283,25.546,154.456
C06049=1076.598,199.189,-77.703,174.281,25.544,154.455
C06050=1076.592,198.941,-77.679,174.279,25.541,154.455
C06051=1076.586,198.692,-77.656,174.276,25.538,154.455
C06052=1076.580,198.443,-77.631,174.274,25.536,154.455
C06053=1076.574,198.194,-77.608,174.271,25.533,154.454
C06054=1076.569,197.945,-77.585,174.269,25.531,154.454
C06055=1076.563,197.696,-77.561,174.267,25.528,154.454
C06056=1076.558,197.448,-77.538,174.264,25.525,154.454
C06057=1076.552,197.199,-77.514,174.263,25.523,154.453
C06058=1076.547,196.950,-77.491,174.261,25.520,154.453
C06059=1076.540,196.702,-77.467,174.258,25.517,154.453
C06060=1076.535,196.452,-77.443,174.256,25.515,154.452
C06061=1076.529,196.204,-77.420,174.253,25.512,154.452
C06062=1076.523,195.955,-77.397,174.251,25.510,154.452
C06063=1076.518,195.705,-77.373,174.249,25.507,154.452
C06064=1076.512,195.457,-77.350,174.246,25.504,154.451
C06065=1076.506,195.208,-77.327,174.245,25.502,154.451
C06066=1076.501,194.959,-77.303,174.243,25.499,154.451
C06067=1076.495,194.711,-77.280,174.240,25.496,154.450
C06068=1076.490,194.462,-77.257,174.238,25.494,154.450
C06069=1076.485,194.213,-77.233,174.236,25.491,154.450
C06070=1076.479,193.964,-77.209,174.233,25.488,154.450
C06071=1076.473,193.716,-77.186,174.232,25.486,154.449
C06072=1076.468,193.466,-77.163,174.229,25.484,154.449
C06073=1076.462,193.217,-77.140,174.227,25.481,154.449
C06074=1076.456,192.969,-77.116,174.225,25.478,154.449
C06075=1076.450,192.719,-77.092,174.222,25.476,154.448
C06076=1076.445,192.470,-77.069,174.220,25.473,154.448
C06077=1076.439,192.221,-77.046,174.218,25.470,154.448
C06078=1076.433,191.973,-77.023,174.216,25.468,154.447
C06079=1076.427,191.692,-76.997,174.213,25.465,154.447
C06080=1076.421,191.412,-76.970,174.211,25.462,154.447
C06081=1076.415,191.131,-76.945,174.208,25.459,154.446
C06082=1076.409,190.850,-76.918,174.206,25.456,154.446
C06083=1076.403,190.602,-76.895,174.204,25.453,154.446
C06084=1076.397,190.353,-76.872,174.201,25.451,154.445
C06085=1076.391,190.104,-76.848,174.199,25.448,154.445
C06086=1076.386,189.855,-76.825,174.197,25.446,154.445
C06087=1076.381,189.606,-76.802,174.195,25.443,154.445
C06088=1076.375,189.357,-76.779,174.193,25.440,154.444
C06089=1076.369,189.109,-76.756,174.190,25.437,154.444
C06090=1076.365,188.860,-76.733,174.188,25.435,154.444
C06091=1076.359,188.611,-76.710,174.187,25.432,154.443
C06092=1076.353,188.362,-76.687,174.184,25.430,154.443
C06093=1076.348,188.113,-76.664,174.182,25.427,154.443
C06094=1076.343,187.864,-76.640,174.180,25.424,154.443
C06095=1076.337,187.615,-76.617,174.177,25.421,154.442
C06096=1076.331,187.366,-76.595,174.176,25.419,154.442
C06097=1076.325,187.117,-76.572,174.173,25.416,154.442
C06098=1076.320,186.869,-76.549,174.171,25.414,154.441
C06099=1076.315,186.620,-76.525,174.169,25.411,154.441
C06100=1076.310,186.371,-76.503,174.167,25.408,154.441
C06101=1076.304,186.122,-76.480,174.165,25.406,154.441
C06102=1076.298,185.873,-76.457,174.163,25.403,154.440
C06103=1076.292,185.624,-76.434,174.160,25.401,154.440
C06104=1076.287,185.375,-76.410,174.158,25.398,154.440
C06105=1076.282,185.126,-76.387,174.156,25.396,154.439
C06106=1076.276,184.878,-76.365,174.154,25.393,154.439
C06107=1076.271,184.629,-76.342,174.152,25.390,154.439
C06108=1076.265,184.380,-76.319,174.149,25.388,154.439
C06109=1076.260,184.131,-76.297,174.148,25.386,154.438
C06110=1076.253,183.882,-76.274,174.146,25.383,154.438
C06111=1076.247,183.633,-76.251,174.143,25.380,154.438
C06112=1076.242,183.384,-76.228,174.141,25.378,154.438
C06113=1076.236,183.136,-76.205,174.139,25.375,154.437
C06114=1076.230,182.887,-76.182,174.137,25.373,154.437
C06115=1076.224,182.637,-76.161,174.135,25.370,154.437
C06116=1076.218,182.389,-76.138,174.132,25.367,154.436
C06117=1076.213,182.140,-76.115,174.131,25.365,154.436
C06118=1076.207,181.891,-76.092,174.128,25.363,154.436
C06119=1076.200,181.642,-76.070,174.126,25.360,154.436
C06120=1076.195,181.393,-76.047,174.124,25.358,154.436
C06121=1076.189,181.144,-76.024,174.122,25.356,154.435
C06122=1076.184,180.896,-76.002,174.120,25.353,154.435
C06123=1076.178,180.646,-75.980,174.117,25.350,154.435
C06124=1076.172,180.397,-75.957,174.115,25.348,154.434
C06125=1076.166,180.149,-75.934,174.114,25.345,154.434
C06126=1076.161,179.900,-75.911,174.111,25.343,154.434
C06127=1076.155,179.650,-75.890,174.109,25.340,154.434
C06128=1076.149,179.402,-75.867,174.107,25.338,154.433
C06129=1076.144,179.153,-75.844,174.105,25.335,154.433
C06130=1076.138,178.904,-75.822,174.103,25.333,154.433
C06131=1076.132,178.655,-75.800,174.100,25.330,154.433
C06132=1076.126,178.406,-75.777,174.098,25.327,154.432
C06133=1076.121,178.157,-75.754,174.097,25.325,154.432
C06134=1076.115,177.908,-75.731,174.094,25.322,154.432
C06135=1076.109,177.659,-75.710,174.092,25.320,154.431
C06136=1076.104,177.411,-75.687,174.090,25.318,154.431
C06137=1076.098,177.161,-75.665,174.088,25.315,154.431
C06138=1076.092,176.912,-75.643,174.086,25.312,154.431
C06139=1076.086,176.664,-75.620,174.083,25.310,154.430
C06140=1076.081,176.415,-75.598,174.082,25.307,154.430
C06141=1076.075,176.166,-75.575,174.080,25.305,154.430
C06142=1076.069,175.917,-75.553,174.077,25.302,154.430
C06143=1076.063,175.636,-75.528,174.075,25.299,154.429
C06144=1076.057,175.355,-75.503,174.073,25.296,154.429
C06145=1076.050,175.074,-75.478,174.070,25.294,154.429
C06146=1076.044,174.793,-75.452,174.068,25.291,154.428
C06147=1076.038,174.544,-75.430,174.066,25.288,154.428
C06148=1076.032,174.295,-75.408,174.064,25.286,154.428
C06149=1076.027,174.046,-75.386,174.062,25.283,154.428
C06150=1076.021,173.797,-75.363,174.059,25.281,154.427
C06151=1076.015,173.548,-75.341,174.058,25.279,154.427
C06152=1076.010,173.299,-75.319,174.056,25.275,154.427
C06153=1076.005,173.050,-75.296,174.053,25.273,154.426
C06154=1075.999,172.801,-75.275,174.052,25.270,154.426
C06155=1075.993,172.553,-75.252,174.050,25.268,154.426
C06156=1075.988,172.303,-75.230,174.047,25.265,154.426
C06157=1075.982,172.054,-75.208,174.046,25.263,154.425
C06158=1075.976,171.805,-75.185,174.043,25.260,154.425
C06159=1075.971,171.556,-75.164,174.041,25.258,154.425
C06160=1075.965,171.307,-75.142,174.040,25.255,154.424
C06161=1075.960,171.059,-75.119,174.037,25.253,154.424
C06162=1075.954,170.810,-75.098,174.035,25.250,154.424
C06163=1075.948,170.560,-75.076,174.034,25.248,154.424
C06164=1075.943,170.312,-75.053,174.031,25.245,154.423
C06165=1075.937,170.063,-75.031,174.029,25.243,154.423
C06166=1075.932,169.813,-75.009,174.027,25.240,154.423
C06167=1075.927,169.565,-74.987,174.025,25.238,154.423
C06168=1075.920,169.316,-74.965,174.023,25.235,154.422
C06169=1075.915,169.067,-74.943,174.021,25.233,154.422
C06170=1075.909,168.818,-74.921,174.019,25.229,154.422
C06171=1075.904,168.568,-74.899,174.017,25.227,154.421
C06172=1075.898,168.321,-74.877,174.015,25.225,154.421
C06173=1075.893,168.071,-74.855,174.013,25.222,154.421
C06174=1075.888,167.822,-74.833,174.011,25.220,154.420
C06175=1075.882,167.573,-74.811,174.009,25.217,154.420
C06176=1075.876,167.324,-74.789,174.007,25.214,154.420
C06177=1075.871,167.075,-74.768,174.005,25.212,154.420
C06178=1075.865,166.826,-74.745,174.003,25.209,154.419
C06179=1075.859,166.578,-74.724,174.001,25.207,154.419
C06180=1075.854,166.328,-74.701,173.999,25.204,154.419
C06181=1075.849,166.079,-74.680,173.997,25.201,154.418
C06182=1075.843,165.830,-74.658,173.996,25.199,154.418
C06183=1075.838,165.581,-74.636,173.993,25.196,154.418
C06184=1075.832,165.332,-74.614,173.991,25.194,154.418
C06185=1075.827,165.083,-74.593,173.989,25.191,154.417
C06186=1075.821,164.834,-74.571,173.987,25.189,154.417
C06187=1075.816,164.586,-74.548,173.985,25.186,154.417
C06188=1075.810,164.337,-74.527,173.983,25.183,154.416
C06189=1075.805,164.088,-74.505,173.981,25.181,154.416
C06190=1075.799,163.839,-74.483,173.980,25.178,154.416
C06191=1075.794,163.590,-74.461,173.977,25.176,154.416
C06192=1075.788,163.341,-74.440,173.975,25.173,154.415
C06193=1075.783,163.092,-74.418,173.973,25.171,154.415
C06194=1075.777,162.843,-74.396,173.971,25.168,154.415
C06195=1075.772,162.594,-74.374,173.970,25.165,154.414
C06196=1075.766,162.345,-74.353,173.968,25.163,154.414
C06197=1075.761,162.096,-74.331,173.965,25.160,154.414
C06198=1075.755,161.847,-74.309,173.964,25.158,154.414
C06199=1075.750,161.598,-74.287,173.961,25.155,154.413
C06200=1075.744,161.348,-74.266,173.960,25.153,154.413
C06201=1075.739,161.099,-74.245,173.958,25.150,154.413
C06202=1075.733,160.850,-74.223,173.955,25.147,154.412
C06203=1075.728,160.601,-74.202,173.954,25.145,154.412
C06204=1075.721,160.352,-74.180,173.951,25.143,154.412
C06205=1075.717,160.103,-74.158,173.950,25.140,154.412
C06206=1075.710,159.854,-74.137,173.948,25.138,154.411
C06207=1075.704,159.573,-74.112,173.946,25.134,154.411
C06208=1075.698,159.291,-74.088,173.943,25.132,154.411
C06209=1075.691,159.010,-74.064,173.941,25.129,154.410
C06210=1075.685,158.729,-74.040,173.939,25.126,154.410
C06211=1075.679,158.480,-74.018,173.937,25.124,154.410
C06212=1075.674,158.231,-73.998,173.935,25.121,154.410
C06213=1075.668,157.982,-73.976,173.933,25.119,154.409
C06214=1075.663,157.733,-73.954,173.931,25.116,154.409
C06215=1075.657,157.484,-73.933,173.930,25.114,154.409
C06216=1075.651,157.235,-73.911,173.927,25.111,154.408
C06217=1075.645,156.985,-73.891,173.925,25.108,154.408
C06218=1075.640,156.737,-73.869,173.924,25.106,154.408
C06219=1075.634,156.488,-73.848,173.921,25.103,154.408
C06220=1075.629,156.238,-73.826,173.920,25.101,154.407
C06221=1075.623,155.990,-73.805,173.918,25.098,154.407
C06222=1075.617,155.741,-73.784,173.916,25.096,154.407
C06223=1075.612,155.492,-73.762,173.914,25.093,154.406
C06224=1075.606,155.242,-73.741,173.912,25.091,154.406
C06225=1075.600,154.994,-73.720,173.910,25.088,154.406
C06226=1075.594,154.745,-73.698,173.908,25.085,154.406
C06227=1075.589,154.495,-73.678,173.906,25.083,154.405
C06228=1075.583,154.247,-73.657,173.904,25.080,154.405
C06229=1075.577,153.998,-73.635,173.903,25.078,154.405
C06230=1075.572,153.749,-73.614,173.900,25.075,154.404
C06231=1075.566,153.499,-73.593,173.899,25.073,154.404
C06232=1075.561,153.250,-73.572,173.896,25.071,154.404
C06233=1075.555,153.002,-73.551,173.895,25.068,154.404
C06234=1075.549,152.753,-73.529,173.893,25.066,154.403
C06235=1075.544,152.503,-73.509,173.891,25.063,154.403
C06236=1075.537,152.254,-73.487,173.889,25.061,154.403
C06237=1075.533,152.005,-73.466,173.887,25.058,154.403
C06238=1075.527,151.756,-73.445,173.885,25.056,154.402
C06239=1075.521,151.507,-73.424,173.883,25.053,154.402
C06240=1075.516,151.258,-73.403,173.881,25.051,154.402
C06241=1075.511,151.009,-73.382,173.879,25.048,154.401
C06242=1075.504,150.760,-73.361,173.878,25.046,154.401
C06243=1075.498,150.511,-73.340,173.875,25.043,154.401
C06244=1075.493,150.262,-73.319,173.874,25.040,154.401
C06245=1075.487,150.013,-73.298,173.872,25.038,154.400
C06246=1075.481,149.764,-73.277,173.870,25.035,154.400
C06247=1075.476,149.515,-73.256,173.868,25.033,154.400
C06248=1075.470,149.266,-73.235,173.866,25.030,154.399
C06249=1075.465,149.017,-73.214,173.864,25.028,154.399
C06250=1075.459,148.768,-73.193,173.863,25.025,154.399
C06251=1075.453,148.518,-73.172,173.860,25.023,154.399
C06252=1075.448,148.269,-73.151,173.859,25.020,154.398
C06253=1075.443,148.021,-73.130,173.857,25.018,154.398
C06254=1075.437,147.771,-73.109,173.855,25.015,154.398
C06255=1075.430,147.523,-73.089,173.853,25.013,154.398
C06256=1075.425,147.273,-73.068,173.851,25.010,154.397
C06257=1075.419,147.024,-73.047,173.849,25.008,154.397
C06258=1075.414,146.775,-73.026,173.848,25.005,154.397
C06259=1075.408,146.526,-73.005,173.845,25.003,154.396
C06260=1075.402,146.277,-72.985,173.844,25.000,154.396
C06261=1075.396,146.028,-72.964,173.842,24.998,154.396
C06262=1075.391,145.779,-72.943,173.840,24.995,154.396
C06263=1075.385,145.529,-72.922,173.838,24.993,154.395
C06264=1075.379,145.281,-72.902,173.836,24.991,154.395
C06265=1075.374,145.032,-72.881,173.834,24.987,154.395
C06266=1075.368,144.783,-72.860,173.833,24.985,154.394
C06267=1075.363,144.533,-72.840,173.831,24.982,154.394
C06268=1075.357,144.284,-72.818,173.829,24.980,154.394
C06269=1075.351,144.035,-72.798,173.827,24.977,154.394
C06270=1075.346,143.786,-72.778,173.825,24.975,154.393
C06271=1075.339,143.505,-72.754,173.823,24.972,154.393
C06272=1075.333,143.223,-72.731,173.821,24.969,154.393
C06273=1075.326,142.941,-72.708,173.819,24.967,154.392
C06274=1075.319,142.660,-72.684,173.817,24.964,154.392
C06275=1075.314,142.410,-72.664,173.815,24.961,154.392
C06276=1075.309,142.161,-72.643,173.814,24.959,154.391
C06277=1075.304,141.912,-72.623,173.811,24.956,154.391
C06278=1075.297,141.663,-72.602,173.810,24.954,154.391
C06279=1075.292,141.414,-72.581,173.807,24.951,154.391
C06280=1075.286,141.165,-72.560,173.806,24.949,154.390
C06281=1075.280,140.916,-72.540,173.804,24.946,154.390
C06282=1075.275,140.667,-72.520,173.802,24.943,154.390
C06283=1075.270,140.418,-72.499,173.800,24.941,154.389
C06284=1075.263,140.169,-72.479,173.799,24.938,154.389
C06285=1075.258,139.919,-72.458,173.796,24.936,154.389
C06286=1075.253,139.670,-72.438,173.795,24.933,154.389
C06287=1075.246,139.422,-72.417,173.793,24.931,154.388
C06288=1075.241,139.172,-72.396,173.791,24.928,154.388
C06289=1075.235,138.923,-72.376,173.790,24.926,154.388
C06290=1075.229,138.674,-72.356,173.787,24.923,154.387
C06291=1075.224,138.425,-72.335,173.786,24.921,154.387
C06292=1075.218,138.176,-72.315,173.784,24.918,154.387
C06293=1075.213,137.927,-72.295,173.782,24.916,154.387
C06294=1075.206,137.678,-72.274,173.780,24.913,154.386
C06295=1075.201,137.429,-72.254,173.779,24.910,154.386
C06296=1075.195,137.180,-72.234,173.776,24.908,154.386
C06297=1075.190,136.931,-72.213,173.775,24.905,154.385
C06298=1075.184,136.682,-72.193,173.774,24.903,154.385
C06299=1075.178,136.433,-72.173,173.771,24.900,154.385
C06300=1075.172,136.183,-72.153,173.770,24.898,154.385
C06301=1075.167,135.934,-72.132,173.768,24.895,154.384
C06302=1075.161,135.685,-72.113,173.766,24.893,154.384
C06303=1075.156,135.436,-72.092,173.764,24.890,154.384
C06304=1075.150,135.187,-72.072,173.762,24.888,154.383
C06305=1075.144,134.938,-72.052,173.760,24.885,154.383
C06306=1075.138,134.689,-72.032,173.759,24.883,154.383
C06307=1075.133,134.440,-72.011,173.757,24.880,154.382
C06308=1075.127,134.190,-71.991,173.755,24.878,154.382
C06309=1075.121,133.941,-71.970,173.754,24.875,154.382
C06310=1075.115,133.692,-71.950,173.751,24.873,154.382
C06311=1075.110,133.442,-71.930,173.750,24.870,154.381
C06312=1075.104,133.194,-71.910,173.748,24.868,154.381
C06313=1075.099,132.945,-71.890,173.746,24.865,154.381
C06314=1075.093,132.696,-71.870,173.745,24.862,154.380
C06315=1075.088,132.447,-71.849,173.743,24.860,154.380
C06316=1075.082,132.197,-71.830,173.741,24.857,154.380
C06317=1075.077,131.948,-71.810,173.739,24.855,154.380
C06318=1075.070,131.699,-71.789,173.737,24.852,154.379
C06319=1075.064,131.450,-71.769,173.736,24.850,154.379
C06320=1075.058,131.201,-71.749,173.734,24.847,154.379
C06321=1075.053,130.951,-71.730,173.732,24.845,154.378
C06322=1075.047,130.702,-71.710,173.730,24.842,154.378
C06323=1075.041,130.454,-71.690,173.729,24.840,154.378
C06324=1075.036,130.204,-71.670,173.726,24.837,154.378
C06325=1075.030,129.955,-71.650,173.725,24.835,154.377
C06326=1075.024,129.706,-71.630,173.723,24.833,154.377
C06327=1075.018,129.457,-71.610,173.721,24.830,154.377
C06328=1075.012,129.207,-71.590,173.720,24.828,154.377
C06329=1075.006,128.958,-71.570,173.717,24.825,154.376
C06330=1075.001,128.709,-71.550,173.716,24.823,154.376
C06331=1074.995,128.460,-71.531,173.715,24.820,154.376
C06332=1074.989,128.211,-71.511,173.712,24.817,154.375
C06333=1074.983,127.962,-71.491,173.711,24.815,154.375
C06334=1074.978,127.713,-71.471,173.709,24.812,154.375
C06335=1074.971,127.430,-71.449,173.707,24.810,154.374
C06336=1074.965,127.150,-71.426,173.705,24.807,154.374
C06337=1074.958,126.868,-71.404,173.703,24.804,154.374
C06338=1074.951,126.586,-71.382,173.702,24.801,154.373
C06339=1074.945,126.337,-71.362,173.699,24.799,154.373
C06340=1074.940,126.087,-71.342,173.698,24.796,154.373
C06341=1074.934,125.838,-71.322,173.696,24.794,154.373
C06342=1074.929,125.589,-71.303,173.694,24.791,154.372
C06343=1074.923,125.340,-71.283,173.693,24.789,154.372
C06344=1074.917,125.091,-71.263,173.690,24.786,154.372
C06345=1074.911,124.842,-71.243,173.689,24.783,154.371
C06346=1074.906,124.593,-71.223,173.688,24.781,154.371
C06347=1074.900,124.343,-71.204,173.685,24.778,154.371
C06348=1074.894,124.094,-71.184,173.684,24.776,154.371
C06349=1074.888,123.845,-71.164,173.682,24.773,154.370
C06350=1074.883,123.597,-71.145,173.680,24.771,154.370
C06351=1074.877,123.347,-71.126,173.679,24.769,154.370
C06352=1074.872,123.098,-71.106,173.677,24.765,154.369
C06353=1074.866,122.849,-71.086,173.675,24.763,154.369
C06354=1074.861,122.599,-71.067,173.674,24.761,154.369
C06355=1074.855,122.351,-71.047,173.672,24.758,154.369
C06356=1074.849,122.101,-71.027,173.670,24.756,154.368
C06357=1074.843,121.852,-71.007,173.668,24.753,154.368
C06358=1074.837,121.603,-70.988,173.667,24.750,154.368
C06359=1074.832,121.353,-70.968,173.665,24.748,154.367
C06360=1074.826,121.104,-70.948,173.663,24.745,154.367
C06361=1074.821,120.855,-70.929,173.662,24.743,154.367
C06362=1074.815,120.606,-70.909,173.660,24.741,154.366
C06363=1074.809,120.357,-70.890,173.658,24.738,154.366
C06364=1074.804,120.108,-70.871,173.657,24.735,154.366
C06365=1074.798,119.859,-70.851,173.655,24.733,154.365
C06366=1074.792,119.610,-70.832,173.653,24.730,154.365
C06367=1074.787,119.360,-70.813,173.652,24.728,154.365
C06368=1074.781,119.111,-70.793,173.650,24.725,154.365
C06369=1074.776,118.862,-70.773,173.648,24.722,154.364
C06370=1074.770,118.612,-70.753,173.647,24.720,154.364
C06371=1074.764,118.363,-70.734,173.644,24.717,154.364
C06372=1074.759,118.115,-70.715,173.643,24.715,154.363
C06373=1074.753,117.865,-70.695,173.642,24.712,154.363
C06374=1074.747,117.616,-70.676,173.639,24.709,154.363
C06375=1074.741,117.367,-70.656,173.638,24.707,154.362
C06376=1074.736,117.118,-70.637,173.637,24.704,154.362
C06377=1074.730,116.868,-70.618,173.634,24.701,154.362
C06378=1074.725,116.619,-70.599,173.633,24.699,154.362
C06379=1074.719,116.371,-70.579,173.632,24.697,154.361
C06380=1074.713,116.121,-70.560,173.629,24.694,154.361
C06381=1074.708,115.872,-70.540,173.628,24.691,154.361
C06382=1074.702,115.622,-70.521,173.627,24.689,154.360
C06383=1074.698,115.373,-70.502,173.624,24.686,154.360
C06384=1074.692,115.124,-70.482,173.623,24.683,154.360
C06385=1074.686,114.875,-70.462,173.622,24.681,154.359
C06386=1074.680,114.626,-70.443,173.619,24.678,154.359
C06387=1074.675,114.376,-70.424,173.618,24.676,154.359
C06388=1074.669,114.127,-70.405,173.617,24.673,154.358
C06389=1074.663,113.878,-70.386,173.614,24.670,154.358
C06390=1074.657,113.629,-70.367,173.613,24.668,154.358
C06391=1074.651,113.380,-70.347,173.612,24.666,154.358
C06392=1074.646,113.131,-70.328,173.609,24.663,154.357
C06393=1074.640,112.881,-70.309,173.608,24.660,154.357
C06394=1074.635,112.632,-70.290,173.607,24.658,154.357
C06395=1074.629,112.383,-70.271,173.604,24.655,154.356
C06396=1074.623,112.134,-70.252,173.603,24.653,154.356
C06397=1074.617,111.884,-70.233,173.602,24.650,154.356
C06398=1074.611,111.635,-70.214,173.599,24.647,154.355
C06399=1074.605,111.354,-70.192,173.598,24.645,154.355
C06400=1074.599,111.072,-70.171,173.596,24.641,154.355
C06401=1074.592,110.790,-70.149,173.595,24.639,154.354
C06402=1074.586,110.509,-70.127,173.592,24.636,154.354
C06403=1074.579,110.259,-70.108,173.591,24.634,154.354
C06404=1074.573,110.010,-70.089,173.589,24.631,154.353
C06405=1074.569,109.761,-70.071,173.587,24.628,154.353
C06406=1074.563,109.511,-70.052,173.586,24.626,154.353
C06407=1074.557,109.262,-70.033,173.584,24.623,154.353
C06408=1074.551,109.013,-70.014,173.582,24.621,154.352
C06409=1074.545,108.763,-69.995,173.581,24.618,154.352
C06410=1074.539,108.515,-69.976,173.580,24.616,154.352
C06411=1074.534,108.265,-69.957,173.577,24.613,154.351
C06412=1074.528,108.016,-69.938,173.576,24.610,154.351
C06413=1074.522,107.767,-69.919,173.575,24.608,154.351
C06414=1074.516,107.518,-69.900,173.572,24.605,154.350
C06415=1074.511,107.269,-69.881,173.571,24.603,154.350
C06416=1074.504,107.019,-69.862,173.570,24.600,154.350
C06417=1074.499,106.770,-69.843,173.567,24.597,154.349
C06418=1074.494,106.521,-69.825,173.566,24.595,154.349
C06419=1074.487,106.272,-69.806,173.565,24.593,154.349
C06420=1074.482,106.022,-69.787,173.563,24.589,154.349
C06421=1074.477,105.773,-69.768,173.561,24.587,154.348
C06422=1074.470,105.524,-69.750,173.560,24.585,154.348
C06423=1074.465,105.275,-69.730,173.558,24.582,154.348
C06424=1074.459,105.025,-69.712,173.556,24.579,154.347
C06425=1074.453,104.776,-69.694,173.555,24.577,154.347
C06426=1074.448,104.527,-69.674,173.553,24.574,154.347
C06427=1074.442,104.278,-69.655,173.551,24.572,154.346
C06428=1074.436,104.029,-69.637,173.550,24.569,154.346
C06429=1074.431,103.779,-69.618,173.549,24.567,154.346
C06430=1074.425,103.530,-69.599,173.547,24.564,154.345
C06431=1074.419,103.281,-69.581,173.545,24.561,154.345
C06432=1074.414,103.032,-69.561,173.544,24.559,154.345
C06433=1074.407,102.782,-69.544,173.542,24.556,154.344
C06434=1074.402,102.533,-69.525,173.540,24.554,154.344
C06435=1074.397,102.284,-69.505,173.539,24.551,154.344
C06436=1074.390,102.035,-69.487,173.537,24.548,154.344
C06437=1074.385,101.785,-69.469,173.536,24.546,154.343
C06438=1074.380,101.536,-69.449,173.534,24.543,154.343
C06439=1074.374,101.288,-69.431,173.532,24.540,154.343
C06440=1074.369,101.037,-69.413,173.531,24.538,154.342
C06441=1074.362,100.788,-69.394,173.529,24.535,154.342
C06442=1074.356,100.539,-69.375,173.527,24.533,154.342
C06443=1074.351,100.290,-69.357,173.526,24.530,154.341
C06444=1074.344,100.041,-69.338,173.525,24.528,154.341
C06445=1074.339,99.791,-69.319,173.522,24.525,154.341
C06446=1074.333,99.542,-69.302,173.521,24.523,154.341
C06447=1074.328,99.293,-69.282,173.520,24.520,154.340
C06448=1074.321,99.043,-69.264,173.518,24.517,154.340
C06449=1074.316,98.795,-69.246,173.516,24.515,154.340
C06450=1074.310,98.545,-69.227,173.515,24.512,154.339
C06451=1074.304,98.296,-69.209,173.513,24.510,154.339
C06452=1074.299,98.047,-69.190,173.511,24.507,154.339
C06453=1074.293,97.797,-69.172,173.510,24.504,154.338
C06454=1074.287,97.549,-69.154,173.508,24.502,154.338
C06455=1074.281,97.299,-69.135,173.507,24.500,154.338
C06456=1074.275,97.049,-69.117,173.505,24.497,154.337
C06457=1074.270,96.801,-69.098,173.504,24.494,154.337
C06458=1074.264,96.551,-69.080,173.502,24.492,154.337
C06459=1074.258,96.303,-69.062,173.501,24.489,154.336
C06460=1074.253,96.053,-69.043,173.499,24.486,154.336
C06461=1074.246,95.803,-69.024,173.497,24.484,154.336
C06462=1074.241,95.554,-69.007,173.496,24.482,154.336
C06463=1074.235,95.272,-68.986,173.494,24.478,154.335
C06464=1074.228,94.991,-68.965,173.493,24.475,154.335
C06465=1074.222,94.709,-68.944,173.490,24.473,154.335
C06466=1074.215,94.427,-68.924,173.489,24.470,154.334
C06467=1074.209,94.178,-68.905,173.487,24.467,154.334
C06468=1074.204,93.929,-68.887,173.486,24.464,154.333
C06469=1074.197,93.680,-68.869,173.484,24.462,154.333
C06470=1074.192,93.430,-68.850,173.483,24.459,154.333
C06471=1074.186,93.181,-68.833,173.481,24.456,154.332
C06472=1074.180,92.932,-68.814,173.479,24.454,154.332
C06473=1074.175,92.682,-68.796,173.478,24.452,154.332
C06474=1074.169,92.434,-68.777,173.477,24.449,154.331
C06475=1074.163,92.184,-68.760,173.474,24.446,154.331
C06476=1074.158,91.935,-68.741,173.473,24.444,154.331
C06477=1074.152,91.686,-68.723,173.472,24.441,154.331
C06478=1074.146,91.437,-68.705,173.470,24.438,154.330
C06479=1074.141,91.186,-68.687,173.468,24.436,154.330
C06480=1074.135,90.938,-68.668,173.467,24.433,154.330
C06481=1074.129,90.688,-68.650,173.466,24.430,154.329
C06482=1074.124,90.439,-68.633,173.464,24.428,154.329
C06483=1074.117,90.190,-68.614,173.462,24.425,154.329
C06484=1074.112,89.940,-68.596,173.461,24.422,154.328
C06485=1074.106,89.691,-68.578,173.459,24.420,154.328
C06486=1074.100,89.441,-68.560,173.458,24.418,154.328
C06487=1074.094,89.193,-68.542,173.457,24.415,154.327
C06488=1074.088,88.943,-68.524,173.454,24.412,154.327
C06489=1074.083,88.694,-68.506,173.453,24.410,154.327
C06490=1074.077,88.444,-68.488,173.452,24.407,154.327
C06491=1074.071,88.196,-68.470,173.450,24.405,154.326
C06492=1074.065,87.946,-68.452,173.448,24.402,154.326
C06493=1074.060,87.697,-68.434,173.447,24.399,154.326
C06494=1074.054,87.447,-68.416,173.445,24.397,154.325
C06495=1074.048,87.198,-68.399,173.444,24.395,154.325
C06496=1074.042,86.949,-68.380,173.442,24.391,154.325
C06497=1074.036,86.700,-68.362,173.441,24.389,154.324
C06498=1074.030,86.450,-68.344,173.439,24.387,154.324
C06499=1074.025,86.201,-68.327,173.438,24.384,154.324
C06500=1074.018,85.951,-68.309,173.436,24.381,154.323
C06501=1074.013,85.703,-68.291,173.434,24.379,154.323
C06502=1074.007,85.454,-68.273,173.433,24.376,154.323
C06503=1074.001,85.204,-68.255,173.432,24.373,154.322
C06504=1073.995,84.955,-68.238,173.430,24.371,154.322
C06505=1073.989,84.705,-68.220,173.428,24.368,154.322
C06506=1073.985,84.456,-68.201,173.427,24.366,154.321
C06507=1073.978,84.206,-68.184,173.425,24.363,154.321
C06508=1073.973,83.957,-68.166,173.424,24.361,154.321
C06509=1073.967,83.708,-68.148,173.422,24.358,154.321
C06510=1073.961,83.458,-68.130,173.421,24.355,154.320
C06511=1073.955,83.210,-68.112,173.419,24.353,154.320
C06512=1073.949,82.960,-68.094,173.418,24.350,154.320
C06513=1073.944,82.711,-68.077,173.417,24.348,154.319
C06514=1073.938,82.462,-68.059,173.414,24.345,154.319
C06515=1073.932,82.212,-68.041,173.413,24.342,154.319
C06516=1073.927,81.963,-68.024,173.412,24.340,154.318
C06517=1073.921,81.714,-68.006,173.410,24.337,154.318
C06518=1073.915,81.465,-67.988,173.409,24.334,154.318
C06519=1073.910,81.216,-67.971,173.407,24.332,154.317
C06520=1073.903,80.966,-67.953,173.406,24.329,154.317
C06521=1073.898,80.717,-67.935,173.404,24.326,154.317
C06522=1073.892,80.467,-67.917,173.403,24.324,154.316
C06523=1073.886,80.218,-67.900,173.401,24.321,154.316
C06524=1073.881,79.969,-67.882,173.399,24.318,154.316
C06525=1073.875,79.719,-67.864,173.398,24.316,154.315
C06526=1073.869,79.470,-67.846,173.397,24.313,154.315
C06527=1073.863,79.188,-67.827,173.395,24.310,154.315
C06528=1073.856,78.907,-67.807,173.393,24.307,154.314
C06529=1073.850,78.625,-67.787,173.391,24.304,154.314
C06530=1073.843,78.343,-67.767,173.390,24.301,154.314
C06531=1073.838,78.094,-67.750,173.389,24.299,154.313
C06532=1073.832,77.845,-67.732,173.387,24.296,154.313
C06533=1073.825,77.595,-67.715,173.385,24.293,154.313
C06534=1073.820,77.346,-67.697,173.384,24.291,154.312
C06535=1073.814,77.097,-67.680,173.382,24.289,154.312
C06536=1073.808,76.847,-67.662,173.381,24.286,154.312
C06537=1073.803,76.598,-67.644,173.379,24.283,154.311
C06538=1073.798,76.349,-67.627,173.378,24.281,154.311
C06539=1073.791,76.099,-67.610,173.376,24.278,154.311
C06540=1073.785,75.850,-67.593,173.375,24.275,154.310
C06541=1073.780,75.601,-67.575,173.374,24.273,154.310
C06542=1073.773,75.351,-67.557,173.372,24.270,154.310
C06543=1073.768,75.102,-67.541,173.370,24.267,154.309
C06544=1073.762,74.853,-67.523,173.369,24.265,154.309
C06545=1073.756,74.603,-67.505,173.368,24.262,154.309
C06546=1073.750,74.354,-67.488,173.366,24.260,154.308
C06547=1073.745,74.105,-67.470,173.364,24.257,154.308
C06548=1073.738,73.855,-67.454,173.363,24.254,154.308
C06549=1073.733,73.606,-67.436,173.361,24.252,154.307
C06550=1073.727,73.357,-67.418,173.360,24.249,154.307
C06551=1073.722,73.107,-67.402,173.359,24.246,154.307
C06552=1073.715,72.858,-67.384,173.357,24.244,154.307
C06553=1073.710,72.609,-67.367,173.355,24.241,154.306
C06554=1073.704,72.360,-67.349,173.354,24.238,154.306
C06555=1073.698,72.110,-67.332,173.353,24.236,154.306
C06556=1073.692,71.861,-67.315,173.351,24.234,154.305
C06557=1073.687,71.612,-67.297,173.350,24.231,154.305
C06558=1073.681,71.362,-67.280,173.348,24.228,154.305
C06559=1073.674,71.113,-67.263,173.347,24.225,154.304
C06560=1073.669,70.864,-67.246,173.345,24.223,154.304
C06561=1073.664,70.614,-67.229,173.344,24.220,154.304
C06562=1073.658,70.365,-67.211,173.343,24.217,154.303
C06563=1073.651,70.116,-67.194,173.340,24.215,154.303
C06564=1073.646,69.866,-67.177,173.339,24.212,154.303
C06565=1073.641,69.617,-67.159,173.338,24.209,154.302
C06566=1073.635,69.367,-67.143,173.337,24.207,154.302
C06567=1073.629,69.118,-67.125,173.335,24.205,154.302
C06568=1073.622,68.869,-67.108,173.333,24.201,154.301
C06569=1073.617,68.619,-67.091,173.332,24.199,154.301
C06570=1073.612,68.370,-67.074,173.330,24.197,154.301
C06571=1073.606,68.121,-67.058,173.329,24.194,154.300
C06572=1073.600,67.871,-67.040,173.328,24.191,154.300
C06573=1073.594,67.622,-67.023,173.326,24.189,154.300
C06574=1073.588,67.373,-67.006,173.324,24.186,154.299
C06575=1073.583,67.123,-66.989,173.323,24.183,154.299
C06576=1073.576,66.874,-66.972,173.322,24.181,154.299
C06577=1073.570,66.625,-66.954,173.320,24.178,154.298
C06578=1073.565,66.375,-66.938,173.319,24.176,154.298
C06579=1073.559,66.126,-66.920,173.318,24.173,154.298
C06580=1073.553,65.877,-66.904,173.316,24.170,154.297
C06581=1073.547,65.627,-66.887,173.314,24.168,154.297
C06582=1073.541,65.378,-66.870,173.313,24.165,154.297
C06583=1073.536,65.128,-66.853,173.312,24.162,154.296
C06584=1073.530,64.879,-66.836,173.310,24.160,154.296
C06585=1073.524,64.630,-66.819,173.308,24.157,154.296
C06586=1073.517,64.380,-66.802,173.307,24.154,154.296
C06587=1073.512,64.131,-66.785,173.306,24.152,154.295
C06588=1073.506,63.882,-66.768,173.304,24.150,154.295
C06589=1073.500,63.633,-66.752,173.303,24.147,154.295
C06590=1073.495,63.383,-66.735,173.302,24.144,154.294
C06591=1073.488,63.101,-66.716,173.300,24.141,154.294
C06592=1073.480,62.819,-66.697,173.298,24.139,154.294
C06593=1073.474,62.538,-66.677,173.296,24.135,154.293
C06594=1073.467,62.256,-66.658,173.295,24.132,154.293
C06595=1073.461,62.006,-66.642,173.294,24.130,154.293
C06596=1073.456,61.757,-66.625,173.291,24.127,154.292
C06597=1073.450,61.508,-66.608,173.290,24.125,154.292
C06598=1073.444,61.259,-66.592,173.289,24.122,154.292
C06599=1073.438,61.008,-66.575,173.287,24.120,154.291
C06600=1073.432,60.760,-66.558,173.286,24.117,154.291
C06601=1073.426,60.510,-66.541,173.285,24.114,154.291
C06602=1073.420,60.261,-66.525,173.283,24.112,154.290
C06603=1073.414,60.012,-66.508,173.281,24.109,154.290
C06604=1073.408,59.762,-66.491,173.280,24.107,154.290
C06605=1073.402,59.512,-66.475,173.279,24.104,154.289
C06606=1073.396,59.263,-66.457,173.277,24.102,154.289
C06607=1073.390,59.014,-66.441,173.276,24.099,154.289
C06608=1073.384,58.765,-66.425,173.274,24.096,154.288
C06609=1073.378,58.515,-66.408,173.273,24.094,154.288
C06610=1073.373,58.266,-66.391,173.271,24.091,154.288
C06611=1073.367,58.017,-66.375,173.270,24.088,154.287
C06612=1073.360,57.767,-66.358,173.269,24.086,154.287
C06613=1073.355,57.517,-66.341,173.267,24.083,154.287
C06614=1073.349,57.268,-66.325,173.266,24.081,154.287
C06615=1073.343,57.019,-66.308,173.264,24.078,154.286
C06616=1073.337,56.770,-66.292,173.262,24.075,154.286
C06617=1073.332,56.520,-66.275,173.261,24.073,154.286
C06618=1073.326,56.271,-66.258,173.260,24.070,154.285
C06619=1073.320,56.021,-66.242,173.259,24.068,154.285
C06620=1073.314,55.773,-66.225,173.257,24.065,154.285
C06621=1073.308,55.523,-66.208,173.255,24.062,154.284
C06622=1073.302,55.274,-66.192,173.254,24.060,154.284
C06623=1073.296,55.024,-66.176,173.252,24.057,154.284
C06624=1073.290,54.774,-66.159,173.251,24.054,154.283
C06625=1073.285,54.525,-66.142,173.250,24.052,154.283
C06626=1073.279,54.275,-66.126,173.249,24.050,154.283
C06627=1073.273,54.026,-66.110,173.246,24.046,154.282
C06628=1073.267,53.777,-66.094,173.245,24.044,154.282
C06629=1073.261,53.528,-66.077,173.244,24.041,154.282
C06630=1073.255,53.278,-66.060,173.243,24.039,154.281
C06631=1073.249,53.029,-66.044,173.241,24.036,154.281
C06632=1073.243,52.780,-66.027,173.240,24.033,154.281
C06633=1073.238,52.530,-66.011,173.239,24.031,154.280
C06634=1073.232,52.281,-65.995,173.236,24.028,154.280
C06635=1073.226,52.031,-65.978,173.235,24.025,154.280
C06636=1073.220,51.782,-65.962,173.234,24.023,154.279
C06637=1073.214,51.532,-65.945,173.233,24.021,154.279
C06638=1073.209,51.283,-65.929,173.231,24.018,154.279
C06639=1073.203,51.034,-65.913,173.230,24.015,154.278
C06640=1073.197,50.784,-65.896,173.229,24.012,154.278
C06641=1073.191,50.535,-65.880,173.227,24.010,154.278
C06642=1073.185,50.285,-65.864,173.225,24.007,154.278
C06643=1073.180,50.036,-65.847,173.224,24.004,154.277
C06644=1073.174,49.787,-65.831,173.223,24.002,154.277
C06645=1073.168,49.537,-65.814,173.222,23.999,154.276
C06646=1073.162,49.288,-65.798,173.220,23.997,154.276
C06647=1073.156,49.038,-65.782,173.219,23.994,154.276
C06648=1073.150,48.789,-65.765,173.217,23.991,154.275
C06649=1073.145,48.540,-65.750,173.215,23.989,154.275
C06650=1073.139,48.291,-65.733,173.214,23.986,154.275
C06651=1073.134,48.041,-65.717,173.213,23.983,154.274
C06652=1073.128,47.791,-65.701,173.212,23.981,154.274
C06653=1073.122,47.542,-65.685,173.210,23.978,154.274
C06654=1073.116,47.293,-65.668,173.209,23.975,154.274
C06655=1073.110,47.011,-65.650,173.207,23.972,154.273
C06656=1073.103,46.728,-65.632,173.206,23.969,154.273
C06657=1073.096,46.447,-65.613,173.204,23.966,154.272
C06658=1073.090,46.164,-65.594,173.203,23.963,154.272
C06659=1073.085,45.916,-65.578,173.201,23.961,154.272
C06660=1073.079,45.666,-65.563,173.200,23.958,154.271
C06661=1073.073,45.416,-65.547,173.198,23.955,154.271
C06662=1073.067,45.167,-65.530,173.196,23.953,154.271
C06663=1073.061,44.918,-65.514,173.195,23.950,154.270
C06664=1073.055,44.668,-65.498,173.194,23.947,154.270
C06665=1073.050,44.418,-65.482,173.193,23.944,154.270
C06666=1073.045,44.169,-65.466,173.191,23.942,154.269
C06667=1073.039,43.920,-65.450,173.190,23.940,154.269
C06668=1073.033,43.671,-65.433,173.189,23.937,154.269
C06669=1073.027,43.421,-65.417,173.187,23.934,154.268
C06670=1073.022,43.171,-65.402,173.185,23.931,154.268
C06671=1073.016,42.922,-65.385,173.184,23.929,154.268
C06672=1073.009,42.673,-65.370,173.183,23.926,154.267
C06673=1073.003,42.424,-65.353,173.181,23.924,154.267
C06674=1072.997,42.174,-65.338,173.180,23.921,154.267
C06675=1072.992,41.924,-65.322,173.179,23.918,154.266
C06676=1072.986,41.676,-65.306,173.177,23.916,154.266
C06677=1072.981,41.426,-65.290,173.176,23.913,154.266
C06678=1072.975,41.176,-65.274,173.174,23.910,154.265
C06679=1072.969,40.927,-65.258,173.173,23.907,154.265
C06680=1072.963,40.677,-65.242,173.172,23.905,154.265
C06681=1072.957,40.428,-65.226,173.170,23.903,154.265
C06682=1072.951,40.178,-65.210,173.169,23.900,154.264
C06683=1072.945,39.929,-65.195,173.168,23.897,154.264
C06684=1072.939,39.680,-65.179,173.166,23.895,154.264
C06685=1072.933,39.431,-65.162,173.164,23.892,154.263
C06686=1072.928,39.181,-65.147,173.163,23.889,154.263
C06687=1072.922,38.931,-65.131,173.162,23.887,154.263
C06688=1072.916,38.682,-65.114,173.161,23.884,154.262
C06689=1072.911,38.433,-65.099,173.159,23.882,154.262
C06690=1072.905,38.183,-65.083,173.158,23.879,154.262
C06691=1072.899,37.933,-65.067,173.156,23.876,154.261
C06692=1072.892,37.684,-65.052,173.154,23.873,154.261
C06693=1072.887,37.435,-65.036,173.153,23.871,154.261
C06694=1072.881,37.185,-65.020,173.152,23.868,154.260
C06695=1072.874,36.936,-65.004,173.151,23.866,154.260
C06696=1072.869,36.687,-64.989,173.149,23.863,154.260
C06697=1072.863,36.437,-64.973,173.148,23.861,154.259
C06698=1072.858,36.187,-64.957,173.147,23.858,154.259
C06699=1072.851,35.938,-64.942,173.145,23.855,154.259
C06700=1072.845,35.688,-64.926,173.143,23.853,154.258
C06701=1072.839,35.439,-64.910,173.142,23.850,154.258
C06702=1072.834,35.190,-64.895,173.141,23.848,154.258
C06703=1072.828,34.941,-64.879,173.139,23.845,154.258
C06704=1072.822,34.691,-64.863,173.138,23.843,154.257
C06705=1072.815,34.442,-64.848,173.137,23.840,154.257
C06706=1072.810,34.192,-64.832,173.136,23.837,154.257
C06707=1072.804,33.943,-64.816,173.133,23.835,154.256
C06708=1072.799,33.693,-64.801,173.132,23.832,154.256
C06709=1072.792,33.444,-64.785,173.131,23.829,154.256
C06710=1072.786,33.194,-64.770,173.130,23.827,154.255
C06711=1072.781,32.945,-64.754,173.128,23.824,154.255
C06712=1072.775,32.696,-64.739,173.127,23.822,154.255
C06713=1072.769,32.446,-64.723,173.126,23.819,154.254
C06714=1072.763,32.197,-64.707,173.124,23.817,154.254
C06715=1072.757,31.947,-64.692,173.123,23.814,154.254
C06716=1072.751,31.698,-64.677,173.121,23.811,154.253
C06717=1072.746,31.448,-64.661,173.120,23.809,154.253
C06718=1072.739,31.199,-64.646,173.118,23.806,154.253
C06719=1072.733,30.917,-64.628,173.117,23.803,154.252
C06720=1072.726,30.635,-64.611,173.115,23.800,154.252
C06721=1072.720,30.353,-64.593,173.114,23.797,154.252
C06722=1072.713,30.071,-64.576,173.113,23.794,154.251
C06723=1072.707,29.821,-64.560,173.110,23.791,154.251
C06724=1072.701,29.571,-64.544,173.109,23.789,154.251
C06725=1072.695,29.323,-64.529,173.108,23.786,154.250
C06726=1072.690,29.073,-64.514,173.107,23.784,154.250
C06727=1072.684,28.823,-64.498,173.105,23.781,154.250
C06728=1072.678,28.573,-64.483,173.104,23.779,154.249
C06729=1072.672,28.325,-64.467,173.103,23.776,154.249
C06730=1072.666,28.075,-64.452,173.102,23.774,154.249
C06731=1072.660,27.825,-64.437,173.100,23.771,154.248
C06732=1072.654,27.577,-64.421,173.098,23.768,154.248
C06733=1072.648,27.327,-64.406,173.097,23.765,154.248
C06734=1072.642,27.077,-64.391,173.095,23.763,154.248
C06735=1072.636,26.827,-64.375,173.094,23.761,154.247
C06736=1072.630,26.579,-64.360,173.093,23.758,154.247
C06737=1072.625,26.329,-64.345,173.092,23.755,154.247
C06738=1072.618,26.079,-64.330,173.090,23.753,154.246
C06739=1072.613,25.830,-64.315,173.089,23.750,154.246
C06740=1072.607,25.580,-64.300,173.087,23.748,154.246
C06741=1072.600,25.331,-64.284,173.086,23.745,154.245
C06742=1072.595,25.082,-64.269,173.084,23.742,154.245
C06743=1072.589,24.832,-64.254,173.083,23.740,154.245
C06744=1072.583,24.582,-64.238,173.082,23.738,154.244
C06745=1072.577,24.333,-64.223,173.081,23.735,154.244
C06746=1072.572,24.084,-64.208,173.079,23.732,154.244
C06747=1072.565,23.834,-64.193,173.078,23.730,154.244
C06748=1072.559,23.585,-64.177,173.077,23.727,154.243
C06749=1072.554,23.336,-64.162,173.074,23.724,154.243
C06750=1072.547,23.086,-64.147,173.073,23.722,154.243
C06751=1072.542,22.836,-64.132,173.072,23.719,154.242
C06752=1072.536,22.587,-64.117,173.071,23.717,154.242
C06753=1072.530,22.337,-64.102,173.069,23.714,154.242
C06754=1072.524,22.088,-64.087,173.068,23.712,154.241
C06755=1072.518,21.838,-64.072,173.067,23.709,154.241
C06756=1072.512,21.588,-64.057,173.065,23.707,154.241
C06757=1072.506,21.340,-64.042,173.064,23.704,154.240
C06758=1072.501,21.090,-64.026,173.063,23.701,154.240
C06759=1072.494,20.840,-64.011,173.061,23.699,154.240
C06760=1072.488,20.592,-63.996,173.059,23.696,154.240
C06761=1072.483,20.342,-63.981,173.058,23.693,154.239
C06762=1072.477,20.093,-63.966,173.057,23.691,154.239
C06763=1072.471,19.843,-63.951,173.056,23.688,154.239
C06764=1072.465,19.593,-63.936,173.054,23.686,154.238
C06765=1072.459,19.344,-63.921,173.053,23.683,154.238
C06766=1072.453,19.094,-63.906,173.052,23.681,154.238
C06767=1072.448,18.845,-63.891,173.050,23.678,154.237
C06768=1072.441,18.595,-63.876,173.048,23.676,154.237
C06769=1072.435,18.346,-63.861,173.047,23.673,154.237
C06770=1072.429,18.097,-63.847,173.046,23.670,154.236
C06771=1072.424,17.847,-63.831,173.044,23.668,154.236
C06772=1072.418,17.597,-63.817,173.043,23.665,154.236
C06773=1072.412,17.348,-63.802,173.042,23.663,154.236
C06774=1072.406,17.098,-63.787,173.040,23.661,154.235
C06775=1072.400,16.849,-63.772,173.039,23.658,154.235
C06776=1072.394,16.599,-63.757,173.038,23.655,154.235
C06777=1072.388,16.350,-63.743,173.036,23.652,154.234
C06778=1072.382,16.100,-63.727,173.034,23.650,154.234
C06779=1072.377,15.851,-63.712,173.033,23.648,154.234
C06780=1072.370,15.602,-63.697,173.032,23.645,154.233
C06781=1072.364,15.352,-63.683,173.031,23.642,154.233
C06782=1072.359,15.103,-63.667,173.029,23.640,154.233
C06783=1072.352,14.821,-63.652,173.028,23.637,154.232
C06784=1072.345,14.541,-63.635,173.026,23.634,154.232
C06785=1072.338,14.260,-63.618,173.025,23.631,154.232
C06786=1072.332,13.980,-63.601,173.023,23.628,154.231
C06787=1072.326,13.730,-63.586,173.021,23.626,154.231
C06788=1072.320,13.481,-63.572,173.020,23.624,154.231
C06789=1072.314,13.231,-63.558,173.019,23.621,154.230
C06790=1072.308,12.982,-63.543,173.018,23.618,154.230
C06791=1072.302,12.733,-63.528,173.016,23.616,154.230
C06792=1072.295,12.483,-63.513,173.015,23.613,154.230
C06793=1072.290,12.234,-63.499,173.014,23.611,154.229
C06794=1072.284,11.984,-63.484,173.012,23.609,154.229
C06795=1072.277,11.734,-63.469,173.011,23.606,154.229
C06796=1072.271,11.485,-63.455,173.009,23.603,154.229
C06797=1072.265,11.235,-63.440,173.007,23.601,154.228
C06798=1072.260,10.986,-63.426,173.006,23.598,154.228
C06799=1072.253,10.736,-63.411,173.005,23.596,154.228
C06800=1072.247,10.487,-63.397,173.004,23.593,154.227
C06801=1072.241,10.237,-63.382,173.002,23.591,154.227
C06802=1072.236,9.988,-63.368,173.001,23.588,154.227
C06803=1072.230,9.738,-63.352,173.000,23.586,154.226
C06804=1072.224,9.489,-63.338,172.998,23.584,154.226
C06805=1072.218,9.239,-63.323,172.997,23.581,154.226
C06806=1072.212,8.990,-63.309,172.995,23.578,154.226
C06807=1072.206,8.740,-63.294,172.994,23.576,154.225
C06808=1072.200,8.491,-63.280,172.992,23.573,154.225
C06809=1072.194,8.241,-63.265,172.991,23.571,154.225
C06810=1072.188,7.992,-63.250,172.990,23.568,154.224
C06811=1072.182,7.742,-63.236,172.988,23.566,154.224
C06812=1072.176,7.493,-63.222,172.987,23.563,154.224
C06813=1072.170,7.243,-63.207,172.986,23.561,154.224
C06814=1072.165,6.994,-63.193,172.985,23.559,154.223
C06815=1072.158,6.744,-63.178,172.983,23.556,154.223
C06816=1072.152,6.495,-63.165,172.981,23.553,154.223
C06817=1072.146,6.245,-63.150,172.980,23.550,154.222
C06818=1072.140,5.995,-63.136,172.979,23.548,154.222
C06819=1072.134,5.746,-63.121,172.977,23.546,154.222
C06820=1072.128,5.497,-63.106,172.976,23.543,154.222
C06821=1072.122,5.247,-63.092,172.975,23.541,154.221
C06822=1072.116,4.998,-63.077,172.973,23.538,154.221
C06823=1072.111,4.748,-63.064,172.972,23.536,154.221
C06824=1072.104,4.498,-63.049,172.971,23.534,154.220
C06825=1072.099,4.249,-63.035,172.969,23.531,154.220
C06826=1072.093,4.000,-63.020,172.967,23.528,154.220
C06827=1072.087,3.750,-63.006,172.966,23.525,154.219
C06828=1072.081,3.501,-62.991,172.965,23.523,154.219
C06829=1072.075,3.250,-62.977,172.963,23.521,154.219
C06830=1072.069,3.001,-62.963,172.962,23.518,154.219
C06831=1072.064,2.752,-62.949,172.961,23.516,154.218
C06832=1072.057,2.502,-62.934,172.960,23.513,154.218
C06833=1072.052,2.253,-62.920,172.958,23.511,154.218
C06834=1072.046,2.004,-62.905,172.957,23.508,154.217
C06835=1072.040,1.753,-62.891,172.956,23.506,154.217
C06836=1072.034,1.504,-62.876,172.953,23.503,154.217
C06837=1072.028,1.255,-62.863,172.952,23.500,154.217
C06838=1072.022,1.005,-62.848,172.951,23.498,154.216
C06839=1072.016,0.756,-62.834,172.950,23.495,154.216
C06840=1072.010,0.506,-62.820,172.948,23.493,154.216
C06841=1072.004,0.257,-62.806,172.947,23.491,154.215
C06842=1071.999,0.007,-62.792,172.946,23.488,154.215
C06843=1071.992,-0.243,-62.777,172.944,23.486,154.215
C06844=1071.987,-0.492,-62.763,172.943,23.483,154.215
C06845=1071.982,-0.742,-62.749,172.942,23.481,154.214
C06846=1071.976,-0.991,-62.734,172.940,23.478,154.214
C06847=1071.968,-1.304,-62.717,172.938,23.475,154.214
C06848=1071.961,-1.617,-62.699,172.936,23.472,154.213
C06849=1071.953,-1.931,-62.681,172.935,23.469,154.213
C06850=1071.946,-2.243,-62.664,172.933,23.466,154.213
C06851=1071.940,-2.492,-62.650,172.932,23.463,154.212
C06852=1071.934,-2.742,-62.635,172.931,23.461,154.212
C06853=1071.928,-2.992,-62.621,172.929,23.458,154.212
C06854=1071.923,-3.241,-62.608,172.928,23.456,154.211
C06855=1071.916,-3.491,-62.593,172.926,23.453,154.211
C06856=1071.910,-3.740,-62.579,172.925,23.451,154.211
C06857=1071.905,-3.990,-62.565,172.923,23.448,154.211
C06858=1071.899,-4.240,-62.551,172.922,23.446,154.210
C06859=1071.892,-4.489,-62.537,172.921,23.443,154.210
C06860=1071.887,-4.738,-62.523,172.919,23.441,154.210
C06861=1071.881,-4.988,-62.509,172.918,23.439,154.209
C06862=1071.874,-5.238,-62.496,172.917,23.436,154.209
C06863=1071.869,-5.487,-62.481,172.915,23.434,154.209
C06864=1071.862,-5.737,-62.468,172.914,23.431,154.209
C06865=1071.856,-5.986,-62.454,172.913,23.429,154.208
C06866=1071.851,-6.236,-62.440,172.911,23.426,154.208
C06867=1071.844,-6.486,-62.426,172.909,23.424,154.208
C06868=1071.838,-6.735,-62.412,172.908,23.421,154.208
C06869=1071.833,-6.984,-62.398,172.907,23.419,154.207
C06870=1071.827,-7.234,-62.385,172.905,23.417,154.207
C06871=1071.821,-7.484,-62.370,172.904,23.415,154.207
C06872=1071.814,-7.733,-62.357,172.903,23.412,154.207
C06873=1071.809,-7.983,-62.343,172.901,23.410,154.206
C06874=1071.802,-8.232,-62.328,172.900,23.407,154.206
C06875=1071.796,-8.482,-62.315,172.899,23.405,154.206
C06876=1071.791,-8.731,-62.301,172.897,23.402,154.205
C06877=1071.785,-8.980,-62.288,172.895,23.400,154.205
C06878=1071.778,-9.231,-62.274,172.894,23.397,154.205
C06879=1071.773,-9.480,-62.260,172.893,23.395,154.205
C06880=1071.767,-9.729,-62.246,172.891,23.392,154.204
C06881=1071.761,-9.979,-62.233,172.890,23.390,154.204
C06882=1071.754,-10.228,-62.218,172.889,23.388,154.204
C06883=1071.749,-10.478,-62.204,172.887,23.385,154.204
C06884=1071.742,-10.727,-62.191,172.886,23.383,154.203
C06885=1071.737,-10.977,-62.177,172.885,23.381,154.203
C06886=1071.732,-11.226,-62.163,172.883,23.378,154.203
C06887=1071.725,-11.476,-62.150,172.881,23.376,154.203
C06888=1071.719,-11.726,-62.136,172.880,23.373,154.202
C06889=1071.713,-11.975,-62.123,172.879,23.371,154.202
C06890=1071.708,-12.225,-62.109,172.877,23.368,154.202
C06891=1071.701,-12.474,-62.095,172.876,23.366,154.201
C06892=1071.695,-12.724,-62.081,172.875,23.364,154.201
C06893=1071.689,-12.974,-62.068,172.873,23.361,154.201
C06894=1071.684,-13.223,-62.054,172.872,23.359,154.201
C06895=1071.677,-13.472,-62.041,172.871,23.356,154.200
C06896=1071.672,-13.722,-62.027,172.869,23.354,154.200
C06897=1071.666,-13.972,-62.013,172.867,23.352,154.200
C06898=1071.660,-14.222,-62.000,172.866,23.349,154.200
C06899=1071.654,-14.454,-61.987,172.865,23.347,154.199
C06900=1071.649,-14.686,-61.974,172.863,23.344,154.199
C06901=1071.643,-14.919,-61.961,172.863,23.343,154.199
C06902=1071.637,-15.151,-61.949,172.861,23.340,154.199
C06903=1071.632,-15.384,-61.937,172.860,23.338,154.198
C06904=1071.627,-15.616,-61.924,172.859,23.336,154.198
C06905=1071.622,-15.848,-61.911,172.857,23.334,154.198
C06906=1071.615,-16.081,-61.899,172.856,23.332,154.198
C06907=1071.610,-16.330,-61.885,172.855,23.329,154.197
C06908=1071.603,-16.580,-61.872,172.853,23.327,154.197
C06909=1071.597,-16.829,-61.858,172.852,23.325,154.197
C06910=1071.592,-17.079,-61.845,172.850,23.322,154.197
C06911=1071.584,-17.356,-61.830,172.849,23.319,154.196
C06912=1071.577,-17.633,-61.816,172.847,23.317,154.196
C06913=1071.572,-17.910,-61.800,172.845,23.314,154.196
C06914=1071.564,-18.187,-61.786,172.844,23.312,154.196
C06915=1071.558,-18.436,-61.772,172.842,23.309,154.195
C06916=1071.553,-18.686,-61.758,172.841,23.307,154.195
C06917=1071.546,-18.935,-61.745,172.840,23.305,154.195
C06918=1071.540,-19.185,-61.732,172.838,23.303,154.195
C06919=1071.534,-19.435,-61.718,172.837,23.300,154.194
C06920=1071.528,-19.685,-61.705,172.836,23.298,154.194
C06921=1071.522,-19.934,-61.692,172.833,23.295,154.194
C06922=1071.517,-20.184,-61.678,172.832,23.293,154.194
C06923=1071.511,-20.433,-61.665,172.831,23.291,154.193
C06924=1071.504,-20.683,-61.652,172.830,23.288,154.193
C06925=1071.499,-20.932,-61.638,172.828,23.286,154.193
C06926=1071.492,-21.182,-61.625,172.827,23.284,154.193
C06927=1071.486,-21.432,-61.612,172.826,23.281,154.192
C06928=1071.480,-21.681,-61.599,172.824,23.279,154.192
C06929=1071.475,-21.931,-61.585,172.823,23.277,154.192
C06930=1071.468,-22.180,-61.572,172.821,23.275,154.192
C06931=1071.462,-22.430,-61.559,172.820,23.272,154.191
C06932=1071.457,-22.680,-61.545,172.818,23.269,154.191
C06933=1071.451,-22.929,-61.532,172.817,23.268,154.191
C06934=1071.445,-23.178,-61.519,172.815,23.265,154.191
C06935=1071.439,-23.428,-61.506,172.814,23.263,154.190
C06936=1071.433,-23.678,-61.492,172.813,23.260,154.190
C06937=1071.427,-23.927,-61.479,172.811,23.258,154.190
C06938=1071.421,-24.177,-61.466,172.810,23.256,154.190
C06939=1071.415,-24.426,-61.453,172.809,23.254,154.189
C06940=1071.409,-24.676,-61.439,172.807,23.251,154.189
C06941=1071.403,-24.926,-61.427,172.806,23.249,154.189
C06942=1071.397,-25.175,-61.414,172.805,23.247,154.189
C06943=1071.391,-25.425,-61.401,172.803,23.244,154.188
C06944=1071.385,-25.675,-61.387,172.801,23.242,154.188
C06945=1071.379,-25.924,-61.373,172.800,23.240,154.188
C06946=1071.373,-26.174,-61.361,172.798,23.237,154.188
C06947=1071.367,-26.423,-61.348,172.797,23.235,154.188
C06948=1071.362,-26.674,-61.335,172.796,23.233,154.187
C06949=1071.356,-26.923,-61.321,172.794,23.231,154.187
C06950=1071.349,-27.172,-61.308,172.793,23.228,154.187
C06951=1071.343,-27.422,-61.295,172.792,23.226,154.187
C06952=1071.337,-27.671,-61.282,172.790,23.224,154.186
C06953=1071.331,-27.921,-61.270,172.789,23.221,154.186
C06954=1071.325,-28.170,-61.256,172.788,23.220,154.186
C06955=1071.319,-28.420,-61.244,172.785,23.217,154.186
C06956=1071.313,-28.670,-61.230,172.784,23.215,154.186
C06957=1071.307,-28.919,-61.218,172.783,23.212,154.185
C06958=1071.301,-29.169,-61.205,172.781,23.210,154.185
C06959=1071.295,-29.419,-61.192,172.780,23.208,154.185
C06960=1071.289,-29.668,-61.179,172.779,23.206,154.185
C06961=1071.283,-29.918,-61.166,172.777,23.204,154.184
C06962=1071.277,-30.167,-61.153,172.776,23.201,154.184
C06963=1071.271,-30.417,-61.140,172.774,23.199,154.184
C06964=1071.264,-30.666,-61.127,172.773,23.197,154.184
C06965=1071.259,-30.916,-61.115,172.772,23.195,154.183
C06966=1071.252,-31.165,-61.101,172.769,23.192,154.183
C06967=1071.246,-31.415,-61.089,172.768,23.190,154.183
C06968=1071.240,-31.664,-61.076,172.767,23.188,154.183
C06969=1071.234,-31.914,-61.063,172.765,23.186,154.183
C06970=1071.228,-32.164,-61.050,172.764,23.184,154.183
C06971=1071.222,-32.413,-61.037,172.763,23.181,154.182
C06972=1071.216,-32.663,-61.025,172.761,23.179,154.182
C06973=1071.210,-32.913,-61.011,172.760,23.177,154.182
C06974=1071.204,-33.162,-60.999,172.759,23.175,154.182
C06975=1071.198,-33.438,-60.985,172.756,23.172,154.181
C06976=1071.192,-33.714,-60.970,172.755,23.170,154.181
C06977=1071.185,-33.991,-60.956,172.754,23.167,154.181
C06978=1071.178,-34.268,-60.942,172.752,23.165,154.181
C06979=1071.172,-34.517,-60.929,172.750,23.162,154.180
C06980=1071.166,-34.767,-60.917,172.749,23.160,154.180
C06981=1071.160,-35.017,-60.904,172.748,23.158,154.180
C06982=1071.154,-35.265,-60.891,172.746,23.156,154.180
C06983=1071.148,-35.515,-60.879,172.745,23.154,154.179
C06984=1071.142,-35.765,-60.866,172.743,23.152,154.179
C06985=1071.136,-36.014,-60.853,172.742,23.149,154.179
C06986=1071.130,-36.264,-60.840,172.741,23.147,154.179
C06987=1071.124,-36.514,-60.828,172.739,23.145,154.179
C06988=1071.118,-36.764,-60.815,172.738,23.143,154.178
C06989=1071.112,-37.013,-60.802,172.737,23.141,154.178
C06990=1071.106,-37.263,-60.789,172.735,23.139,154.178
C06991=1071.101,-37.512,-60.777,172.733,23.136,154.178
C06992=1071.095,-37.761,-60.764,172.732,23.134,154.178
C06993=1071.089,-38.011,-60.751,172.730,23.132,154.177
C06994=1071.083,-38.261,-60.739,172.729,23.130,154.177
C06995=1071.077,-38.511,-60.726,172.727,23.127,154.177
C06996=1071.070,-38.761,-60.714,172.726,23.125,154.177
C06997=1071.064,-39.010,-60.701,172.725,23.123,154.177
C06998=1071.059,-39.259,-60.689,172.723,23.121,154.176
C06999=1071.053,-39.509,-60.676,172.722,23.119,154.176
C07000=1071.046,-39.759,-60.664,172.721,23.117,154.176
C07001=1071.040,-40.008,-60.652,172.719,23.115,154.176
C07002=1071.034,-40.258,-60.638,172.718,23.112,154.176
C07003=1071.028,-40.508,-60.626,172.715,23.110,154.175
C07004=1071.022,-40.757,-60.614,172.714,23.108,154.175
C07005=1071.016,-41.007,-60.601,172.713,23.106,154.175
C07006=1071.010,-41.257,-60.589,172.711,23.104,154.175
C07007=1071.005,-41.506,-60.577,172.710,23.102,154.175
C07008=1070.998,-41.755,-60.564,172.709,23.100,154.174
C07009=1070.992,-42.005,-60.551,172.707,23.098,154.174
C07010=1070.986,-42.255,-60.539,172.706,23.095,154.174
C07011=1070.980,-42.505,-60.526,172.704,23.093,154.174
C07012=1070.973,-42.754,-60.514,172.703,23.092,154.174
C07013=1070.968,-43.003,-60.502,172.702,23.089,154.173
C07014=1070.962,-43.253,-60.490,172.700,23.087,154.173
C07015=1070.956,-43.503,-60.477,172.699,23.085,154.173
C07016=1070.949,-43.753,-60.465,172.697,23.082,154.173
C07017=1070.944,-44.003,-60.453,172.695,23.081,154.173
C07018=1070.938,-44.253,-60.440,172.694,23.079,154.173
C07019=1070.931,-44.501,-60.428,172.692,23.076,154.172
C07020=1070.925,-44.751,-60.415,172.691,23.074,154.172
C07021=1070.919,-45.001,-60.403,172.690,23.073,154.172
C07022=1070.913,-45.250,-60.391,172.688,23.070,154.172
C07023=1070.907,-45.500,-60.378,172.687,23.068,154.172
C07024=1070.902,-45.749,-60.366,172.685,23.066,154.171
C07025=1070.896,-45.999,-60.353,172.684,23.064,154.171
C07026=1070.889,-46.249,-60.341,172.683,23.062,154.171
C07027=1070.883,-46.499,-60.329,172.681,23.060,154.171
C07028=1070.878,-46.748,-60.317,172.679,23.058,154.171
C07029=1070.871,-46.997,-60.305,172.678,23.055,154.170
C07030=1070.865,-47.247,-60.292,172.676,23.054,154.170
C07031=1070.859,-47.497,-60.280,172.675,23.052,154.170
C07032=1070.853,-47.746,-60.268,172.673,23.049,154.170
C07033=1070.848,-47.996,-60.256,172.672,23.047,154.170
C07034=1070.842,-48.246,-60.244,172.670,23.045,154.170
C07035=1070.835,-48.496,-60.232,172.669,23.044,154.169
C07036=1070.830,-48.745,-60.219,172.668,23.041,154.169
C07037=1070.824,-48.995,-60.207,172.666,23.039,154.169
C07038=1070.817,-49.245,-60.195,172.665,23.037,154.169
C07039=1070.811,-49.522,-60.181,172.663,23.034,154.169
C07040=1070.805,-49.798,-60.168,172.661,23.033,154.169
C07041=1070.798,-50.075,-60.154,172.660,23.030,154.168
C07042=1070.791,-50.351,-60.141,172.658,23.028,154.168
C07043=1070.785,-50.601,-60.129,172.656,23.026,154.168
C07044=1070.779,-50.851,-60.117,172.655,23.024,154.168
C07045=1070.773,-51.100,-60.105,172.653,23.022,154.168
C07046=1070.767,-51.349,-60.093,172.652,23.020,154.167
C07047=1070.760,-51.599,-60.081,172.651,23.018,154.167
C07048=1070.753,-51.849,-60.069,172.649,23.016,154.167
C07049=1070.748,-52.098,-60.057,172.648,23.014,154.167
C07050=1070.742,-52.348,-60.045,172.646,23.012,154.167
C07051=1070.736,-52.598,-60.033,172.645,23.010,154.167
C07052=1070.729,-52.847,-60.021,172.643,23.008,154.167
C07053=1070.723,-53.096,-60.009,172.642,23.007,154.166
C07054=1070.718,-53.347,-59.997,172.640,23.005,154.166
C07055=1070.711,-53.596,-59.985,172.639,23.003,154.166
C07056=1070.704,-53.846,-59.973,172.637,23.001,154.166
C07057=1070.699,-54.095,-59.961,172.635,22.999,154.166
C07058=1070.693,-54.345,-59.950,172.634,22.997,154.166
C07059=1070.686,-54.595,-59.938,172.632,22.995,154.166
C07060=1070.680,-54.845,-59.925,172.631,22.993,154.165
C07061=1070.674,-55.094,-59.914,172.630,22.991,154.165
C07062=1070.668,-55.344,-59.902,172.628,22.989,154.165
C07063=1070.662,-55.594,-59.890,172.627,22.987,154.165
C07064=1070.656,-55.843,-59.878,172.625,22.985,154.165
C07065=1070.650,-56.092,-59.866,172.624,22.983,154.165
C07066=1070.643,-56.343,-59.855,172.622,22.981,154.164
C07067=1070.637,-56.591,-59.843,172.621,22.979,154.164
C07068=1070.631,-56.841,-59.831,172.619,22.977,154.164
C07069=1070.625,-57.092,-59.819,172.618,22.975,154.164
C07070=1070.619,-57.340,-59.808,172.617,22.974,154.164
C07071=1070.612,-57.590,-59.796,172.615,22.972,154.164
C07072=1070.607,-57.841,-59.784,172.613,22.969,154.164
C07073=1070.601,-58.089,-59.772,172.611,22.967,154.163
C07074=1070.594,-58.339,-59.760,172.610,22.966,154.163
C07075=1070.589,-58.589,-59.748,172.608,22.964,154.163
C07076=1070.582,-58.838,-59.737,172.607,22.962,154.163
C07077=1070.576,-59.089,-59.726,172.606,22.960,154.163
C07078=1070.570,-59.338,-59.713,172.604,22.958,154.163
C07079=1070.564,-59.587,-59.701,172.602,22.957,154.163
C07080=1070.558,-59.837,-59.690,172.601,22.955,154.162
C07081=1070.551,-60.087,-59.678,172.600,22.953,154.162
C07082=1070.546,-60.337,-59.667,172.598,22.951,154.162
C07083=1070.540,-60.586,-59.655,172.597,22.949,154.162
C07084=1070.534,-60.835,-59.643,172.595,22.947,154.162
C07085=1070.528,-61.086,-59.631,172.594,22.945,154.162
C07086=1070.521,-61.335,-59.619,172.592,22.943,154.162
C07087=1070.516,-61.585,-59.609,172.590,22.941,154.161
C07088=1070.509,-61.834,-59.597,172.589,22.939,154.161
C07089=1070.504,-62.084,-59.585,172.587,22.937,154.161
C07090=1070.497,-62.334,-59.573,172.586,22.935,154.161
C07091=1070.491,-62.584,-59.562,172.584,22.934,154.161
C07092=1070.485,-62.833,-59.550,172.583,22.932,154.161
C07093=1070.479,-63.083,-59.539,172.581,22.930,154.161
C07094=1070.473,-63.332,-59.527,172.580,22.928,154.160
C07095=1070.467,-63.582,-59.516,172.578,22.927,154.160
C07096=1070.461,-63.831,-59.504,172.577,22.925,154.160
C07097=1070.455,-64.082,-59.492,172.575,22.923,154.160
C07098=1070.449,-64.331,-59.481,172.574,22.921,154.160
C07099=1070.443,-64.581,-59.469,172.572,22.919,154.160
C07100=1070.437,-64.830,-59.458,172.571,22.917,154.160
C07101=1070.431,-65.080,-59.446,172.570,22.915,154.160
C07102=1070.425,-65.330,-59.434,172.568,22.913,154.159
C07103=1070.418,-65.608,-59.422,172.566,22.911,154.159
C07104=1070.411,-65.886,-59.409,172.564,22.909,154.159
C07105=1070.405,-66.163,-59.396,172.563,22.907,154.159
C07106=1070.398,-66.442,-59.383,172.561,22.905,154.159
C07107=1070.392,-66.691,-59.372,172.559,22.903,154.159
C07108=1070.386,-66.941,-59.360,172.558,22.901,154.159
C07109=1070.380,-67.190,-59.349,172.556,22.899,154.158
C07110=1070.374,-67.440,-59.338,172.555,22.898,154.158
C07111=1070.368,-67.690,-59.326,172.553,22.896,154.158
C07112=1070.362,-67.940,-59.314,172.552,22.894,154.158
C07113=1070.356,-68.189,-59.304,172.550,22.892,154.158
C07114=1070.350,-68.439,-59.292,172.549,22.890,154.158
C07115=1070.344,-68.688,-59.281,172.547,22.889,154.158
C07116=1070.339,-68.938,-59.269,172.546,22.887,154.158
C07117=1070.332,-69.188,-59.257,172.544,22.885,154.158
C07118=1070.327,-69.437,-59.246,172.543,22.883,154.157
C07119=1070.320,-69.687,-59.235,172.541,22.882,154.157
C07120=1070.314,-69.936,-59.224,172.540,22.880,154.157
C07121=1070.308,-70.187,-59.212,172.538,22.878,154.157
C07122=1070.303,-70.436,-59.201,172.537,22.876,154.157
C07123=1070.296,-70.686,-59.189,172.536,22.874,154.157
C07124=1070.290,-70.935,-59.178,172.534,22.873,154.157
C07125=1070.285,-71.185,-59.167,172.532,22.870,154.157
C07126=1070.278,-71.435,-59.156,172.530,22.869,154.157
C07127=1070.272,-71.684,-59.144,172.529,22.867,154.156
C07128=1070.267,-71.934,-59.133,172.527,22.865,154.156
C07129=1070.261,-72.184,-59.122,172.526,22.863,154.156
C07130=1070.255,-72.433,-59.111,172.524,22.862,154.156
C07131=1070.249,-72.683,-59.099,172.523,22.860,154.156
C07132=1070.243,-72.932,-59.088,172.521,22.858,154.156
C07133=1070.236,-73.183,-59.077,172.520,22.856,154.156
C07134=1070.231,-73.432,-59.066,172.518,22.855,154.156
C07135=1070.226,-73.682,-59.054,172.517,22.853,154.155
C07136=1070.219,-73.932,-59.042,172.515,22.851,154.155
C07137=1070.213,-74.181,-59.031,172.514,22.849,154.155
C07138=1070.207,-74.431,-59.020,172.512,22.848,154.155
C07139=1070.201,-74.681,-59.009,172.511,22.846,154.155
C07140=1070.196,-74.930,-58.998,172.509,22.845,154.155
C07141=1070.189,-75.180,-58.987,172.508,22.843,154.155
C07142=1070.183,-75.430,-58.977,172.506,22.841,154.155
C07143=1070.176,-75.679,-58.965,172.505,22.840,154.155
C07144=1070.170,-75.929,-58.954,172.503,22.838,154.155
C07145=1070.165,-76.178,-58.943,172.502,22.836,154.155
C07146=1070.158,-76.428,-58.932,172.500,22.834,154.154
C07147=1070.152,-76.678,-58.921,172.499,22.833,154.154
C07148=1070.146,-76.928,-58.910,172.496,22.831,154.154
C07149=1070.140,-77.177,-58.899,172.495,22.829,154.154
C07150=1070.135,-77.427,-58.888,172.493,22.828,154.154
C07151=1070.128,-77.677,-58.877,172.492,22.826,154.154
C07152=1070.123,-77.927,-58.866,172.490,22.824,154.154
C07153=1070.116,-78.176,-58.854,172.489,22.822,154.154
C07154=1070.109,-78.425,-58.844,172.487,22.821,154.154
C07155=1070.104,-78.675,-58.833,172.486,22.819,154.154
C07156=1070.097,-78.925,-58.822,172.484,22.818,154.154
C07157=1070.092,-79.175,-58.811,172.483,22.816,154.153
C07158=1070.086,-79.424,-58.800,172.481,22.815,154.153
C07159=1070.080,-79.674,-58.789,172.480,22.813,154.153
C07160=1070.074,-79.924,-58.778,172.478,22.811,154.153
C07161=1070.067,-80.173,-58.767,172.477,22.809,154.153
C07162=1070.061,-80.423,-58.756,172.475,22.808,154.153
C07163=1070.055,-80.673,-58.745,172.473,22.807,154.153
C07164=1070.049,-80.923,-58.734,172.472,22.805,154.153
C07165=1070.042,-81.172,-58.724,172.470,22.804,154.153
C07166=1070.037,-81.421,-58.713,172.469,22.802,154.153
C07167=1070.030,-81.702,-58.701,172.467,22.800,154.153
C07168=1070.023,-81.982,-58.689,172.465,22.798,154.153
C07169=1070.016,-82.262,-58.676,172.463,22.797,154.153
C07170=1070.009,-82.542,-58.665,172.462,22.795,154.153
C07171=1070.003,-82.792,-58.653,172.460,22.793,154.152
C07172=1069.997,-83.042,-58.642,172.459,22.792,154.152
C07173=1069.990,-83.291,-58.632,172.457,22.790,154.152
C07174=1069.984,-83.542,-58.622,172.456,22.789,154.152
C07175=1069.979,-83.791,-58.611,172.454,22.788,154.152
C07176=1069.972,-84.040,-58.601,172.452,22.786,154.152
C07177=1069.966,-84.291,-58.589,172.451,22.784,154.152
C07178=1069.960,-84.540,-58.578,172.449,22.783,154.152
C07179=1069.954,-84.789,-58.568,172.448,22.781,154.152
C07180=1069.947,-85.039,-58.557,172.445,22.779,154.152
C07181=1069.941,-85.289,-58.546,172.444,22.778,154.152
C07182=1069.935,-85.539,-58.536,172.442,22.777,154.152
C07183=1069.929,-85.789,-58.525,172.441,22.775,154.152
C07184=1069.923,-86.038,-58.514,172.439,22.773,154.152
C07185=1069.917,-86.288,-58.504,172.437,22.772,154.152
C07186=1069.911,-86.537,-58.493,172.436,22.770,154.152
C07187=1069.904,-86.787,-58.483,172.434,22.769,154.152
C07188=1069.898,-87.037,-58.472,172.433,22.768,154.152
C07189=1069.893,-87.287,-58.461,172.431,22.766,154.152
C07190=1069.886,-87.536,-58.451,172.430,22.764,154.151
C07191=1069.880,-87.786,-58.440,172.428,22.763,154.151
C07192=1069.874,-88.035,-58.429,172.426,22.762,154.151
C07193=1069.868,-88.285,-58.419,172.425,22.760,154.151
C07194=1069.862,-88.535,-58.408,172.423,22.758,154.151
C07195=1069.856,-88.785,-58.397,172.422,22.757,154.151
C07196=1069.849,-89.034,-58.387,172.420,22.756,154.151
C07197=1069.844,-89.284,-58.377,172.419,22.754,154.151
C07198=1069.837,-89.534,-58.366,172.417,22.753,154.151
C07199=1069.831,-89.784,-58.355,172.416,22.751,154.151
C07200=1069.825,-90.033,-58.345,172.414,22.750,154.151
C07201=1069.819,-90.283,-58.335,172.412,22.748,154.151
C07202=1069.814,-90.532,-58.324,172.411,22.747,154.151
C07203=1069.806,-90.782,-58.313,172.409,22.746,154.151
C07204=1069.801,-91.032,-58.303,172.408,22.744,154.151
C07205=1069.795,-91.282,-58.292,172.406,22.742,154.151
C07206=1069.789,-91.531,-58.282,172.404,22.741,154.151
C07207=1069.783,-91.781,-58.272,172.403,22.740,154.151
C07208=1069.776,-92.031,-58.261,172.401,22.738,154.151
C07209=1069.771,-92.280,-58.250,172.400,22.737,154.151
C07210=1069.765,-92.531,-58.240,172.398,22.735,154.151
C07211=1069.759,-92.780,-58.230,172.396,22.734,154.151
C07212=1069.753,-93.029,-58.219,172.395,22.733,154.151
C07213=1069.747,-93.279,-58.210,172.393,22.731,154.151
C07214=1069.740,-93.529,-58.198,172.392,22.730,154.151
C07215=1069.734,-93.779,-58.189,172.390,22.729,154.151
C07216=1069.728,-94.029,-58.178,172.388,22.727,154.151
C07217=1069.723,-94.278,-58.167,172.387,22.725,154.150
C07218=1069.717,-94.528,-58.157,172.385,22.724,154.150
C07219=1069.711,-94.777,-58.147,172.384,22.723,154.150
C07220=1069.704,-95.028,-58.137,172.382,22.721,154.150
C07221=1069.698,-95.277,-58.126,172.381,22.720,154.150
C07222=1069.692,-95.526,-58.115,172.379,22.719,154.150
C07223=1069.686,-95.777,-58.105,172.377,22.717,154.150
C07224=1069.680,-96.026,-58.095,172.376,22.716,154.150
C07225=1069.674,-96.276,-58.085,172.374,22.715,154.150
C07226=1069.669,-96.525,-58.074,172.372,22.713,154.150
C07227=1069.663,-96.775,-58.064,172.371,22.712,154.150
C07228=1069.657,-97.025,-58.054,172.369,22.710,154.150
C07229=1069.650,-97.275,-58.044,172.368,22.709,154.150
C07230=1069.644,-97.525,-58.033,172.366,22.707,154.150
C07231=1069.638,-97.807,-58.021,172.365,22.706,154.150
C07232=1069.630,-98.090,-58.010,172.362,22.704,154.150
C07233=1069.623,-98.372,-57.999,172.360,22.703,154.150
C07234=1069.617,-98.654,-57.988,172.359,22.702,154.150
C07235=1069.610,-98.903,-57.977,172.357,22.700,154.150
C07236=1069.604,-99.154,-57.967,172.356,22.699,154.150
C07237=1069.598,-99.403,-57.957,172.354,22.698,154.150
C07238=1069.592,-99.653,-57.947,172.352,22.697,154.150
C07239=1069.586,-99.903,-57.936,172.351,22.695,154.150
C07240=1069.580,-100.152,-57.927,172.349,22.694,154.150
C07241=1069.573,-100.402,-57.916,172.347,22.693,154.150
C07242=1069.568,-100.652,-57.906,172.346,22.691,154.150
C07243=1069.562,-100.901,-57.897,172.344,22.690,154.150
C07244=1069.554,-101.151,-57.886,172.343,22.689,154.150
C07245=1069.549,-101.401,-57.876,172.341,22.688,154.150
C07246=1069.543,-101.651,-57.865,172.339,22.687,154.150
C07247=1069.536,-101.900,-57.856,172.337,22.685,154.150
C07248=1069.531,-102.151,-57.846,172.336,22.684,154.150
C07249=1069.524,-102.400,-57.835,172.334,22.683,154.150
C07250=1069.518,-102.650,-57.826,172.333,22.681,154.150
C07251=1069.513,-102.899,-57.815,172.331,22.680,154.150
C07252=1069.506,-103.149,-57.805,172.329,22.679,154.150
C07253=1069.500,-103.399,-57.796,172.328,22.678,154.150
C07254=1069.494,-103.648,-57.786,172.326,22.676,154.150
C07255=1069.488,-103.898,-57.775,172.324,22.675,154.150
C07256=1069.482,-104.148,-57.766,172.323,22.674,154.150
C07257=1069.476,-104.397,-57.756,172.321,22.673,154.150
C07258=1069.470,-104.648,-57.745,172.319,22.672,154.150
C07259=1069.463,-104.897,-57.735,172.318,22.670,154.150
C07260=1069.457,-105.147,-57.726,172.316,22.669,154.150
C07261=1069.451,-105.396,-57.716,172.314,22.668,154.150
C07262=1069.445,-105.647,-57.705,172.313,22.667,154.150
C07263=1069.439,-105.896,-57.696,172.311,22.665,154.150
C07264=1069.433,-106.146,-57.686,172.310,22.664,154.150
